   DATA[2295,34] := 2.0;
   DATA[2295,35] := 250.1762;
   DATA[2295,36] := 1.681991;
   DATA[2295,37] := 189.1022;
   DATA[2295,38] := 0.000128152;
   DATA[2295,39] := 1.0;
   DATA[2295,40] := 1.0;
   DATA[2296,0] := 2.444992;
   DATA[2296,1] := 865.3663;
   DATA[2296,2] := 2.0;
   DATA[2296,3] := 2.0;
   DATA[2296,4] := 262.3366;
   DATA[2296,5] := 8.395475;
   DATA[2296,6] := 330.0948;
   DATA[2296,7] := 2.455259;
   DATA[2296,8] := 2.0;
   DATA[2296,9] := 2.0;
   DATA[2296,10] := 2.0;
   DATA[2296,11] := 19.70037;
   DATA[2296,12] := 2.203632;
   DATA[2296,13] := 815.7364;
   DATA[2296,14] := 1.0;
   DATA[2296,15] := 2.0;
   DATA[2296,16] := 1.0;
   DATA[2296,17] := 1.0;
   DATA[2296,18] := 1.0;
   DATA[2296,19] := 2.0;
   DATA[2296,20] := 148.808;
   DATA[2296,21] := 155.0115;
   DATA[2296,22] := 1.714926;
   DATA[2296,23] := 851.2817;
   DATA[2296,24] := 2.0;
   DATA[2296,25] := 2.0;
   DATA[2296,26] := 7.873174;
   DATA[2296,27] := 144.3989;
   DATA[2296,28] := 261.7278;
   DATA[2296,29] := 11.95847;
   DATA[2296,30] := 1.723148;
   DATA[2296,31] := 1.281798;
   DATA[2296,32] := 0.7348846;
   DATA[2296,33] := 0.3083624;
   DATA[2296,34] := 2.0;
   DATA[2296,35] := 250.1762;
   DATA[2296,36] := 1.681991;
   DATA[2296,37] := 188.958;
   DATA[2296,38] := 0.000128152;
   DATA[2296,39] := 1.0;
   DATA[2296,40] := 1.0;
   DATA[2297,0] := 2.431861;
   DATA[2297,1] := 865.1308;
   DATA[2297,2] := 2.0;
   DATA[2297,3] := 2.0;
   DATA[2297,4] := 262.3366;
   DATA[2297,5] := 8.395475;
   DATA[2297,6] := 330.0948;
   DATA[2297,7] := 2.455259;
   DATA[2297,8] := 2.0;
   DATA[2297,9] := 2.0;
   DATA[2297,10] := 2.0;
   DATA[2297,11] := 19.70037;
   DATA[2297,12] := 2.203632;
   DATA[2297,13] := 815.456;
   DATA[2297,14] := 1.0;
   DATA[2297,15] := 2.0;
   DATA[2297,16] := 1.0;
   DATA[2297,17] := 1.0;
   DATA[2297,18] := 1.0;
   DATA[2297,19] := 2.0;
   DATA[2297,20] := 148.808;
   DATA[2297,21] := 155.0115;
   DATA[2297,22] := 1.714926;
   DATA[2297,23] := 851.2433;
   DATA[2297,24] := 2.0;
   DATA[2297,25] := 2.0;
   DATA[2297,26] := 7.873174;
   DATA[2297,27] := 144.3989;
   DATA[2297,28] := 261.7278;
   DATA[2297,29] := 11.95847;
   DATA[2297,30] := 1.723148;
   DATA[2297,31] := 1.304214;
   DATA[2297,32] := 0.7348846;
   DATA[2297,33] := 0.3083624;
   DATA[2297,34] := 2.0;
   DATA[2297,35] := 250.1762;
   DATA[2297,36] := 1.681991;
   DATA[2297,37] := 188.958;
   DATA[2297,38] := 0.000128152;
   DATA[2297,39] := 1.0;
   DATA[2297,40] := 1.0;
   DATA[2298,0] := 2.425776;
   DATA[2298,1] := 865.4056;
   DATA[2298,2] := 2.0;
   DATA[2298,3] := 2.0;
   DATA[2298,4] := 262.3366;
   DATA[2298,5] := 8.395475;
   DATA[2298,6] := 330.0948;
   DATA[2298,7] := 2.455259;
   DATA[2298,8] := 2.0;
   DATA[2298,9] := 2.0;
   DATA[2298,10] := 2.0;
   DATA[2298,11] := 19.70037;
   DATA[2298,12] := 2.203632;
   DATA[2298,13] := 815.6162;
   DATA[2298,14] := 1.0;
   DATA[2298,15] := 2.0;
   DATA[2298,16] := 1.0;
   DATA[2298,17] := 1.0;
   DATA[2298,18] := 1.0;
   DATA[2298,19] := 2.0;
   DATA[2298,20] := 148.808;
   DATA[2298,21] := 155.0115;
   DATA[2298,22] := 1.714926;
   DATA[2298,23] := 851.3971;
   DATA[2298,24] := 2.0;
   DATA[2298,25] := 2.0;
   DATA[2298,26] := 7.873174;
   DATA[2298,27] := 144.3989;
   DATA[2298,28] := 261.7278;
   DATA[2298,29] := 11.95847;
   DATA[2298,30] := 1.723148;
   DATA[2298,31] := 1.310747;
   DATA[2298,32] := 0.7348846;
   DATA[2298,33] := 0.3083624;
   DATA[2298,34] := 2.0;
   DATA[2298,35] := 250.1762;
   DATA[2298,36] := 1.681991;
   DATA[2298,37] := 188.958;
   DATA[2298,38] := 0.000128152;
   DATA[2298,39] := 1.0;
   DATA[2298,40] := 1.0;
   DATA[2299,0] := 2.425456;
   DATA[2299,1] := 865.5626;
   DATA[2299,2] := 2.0;
   DATA[2299,3] := 2.0;
   DATA[2299,4] := 262.3366;
   DATA[2299,5] := 8.395475;
   DATA[2299,6] := 330.0948;
   DATA[2299,7] := 2.456156;
   DATA[2299,8] := 2.0;
   DATA[2299,9] := 2.0;
   DATA[2299,10] := 2.0;
   DATA[2299,11] := 19.67796;
   DATA[2299,12] := 2.206322;
   DATA[2299,13] := 815.416;
   DATA[2299,14] := 1.0;
   DATA[2299,15] := 2.0;
   DATA[2299,16] := 1.0;
   DATA[2299,17] := 1.0;
   DATA[2299,18] := 1.0;
   DATA[2299,19] := 2.0;
   DATA[2299,20] := 148.808;
   DATA[2299,21] := 155.0115;
   DATA[2299,22] := 1.714926;
   DATA[2299,23] := 851.3971;
   DATA[2299,24] := 2.0;
   DATA[2299,25] := 2.0;
   DATA[2299,26] := 7.874776;
   DATA[2299,27] := 144.5014;
   DATA[2299,28] := 261.7278;
   DATA[2299,29] := 11.95847;
   DATA[2299,30] := 1.725327;
   DATA[2299,31] := 1.311772;
   DATA[2299,32] := 0.7348846;
   DATA[2299,33] := 0.3083624;
   DATA[2299,34] := 2.0;
   DATA[2299,35] := 250.1762;
   DATA[2299,36] := 1.681991;
   DATA[2299,37] := 188.958;
   DATA[2299,38] := 0.000128152;
   DATA[2299,39] := 1.0;
   DATA[2299,40] := 1.0;
   DATA[2300,0] := 2.451398;
   DATA[2300,1] := 865.7589;
   DATA[2300,2] := 2.0;
   DATA[2300,3] := 2.0;
   DATA[2300,4] := 262.3366;
   DATA[2300,5] := 8.395475;
   DATA[2300,6] := 330.0948;
   DATA[2300,7] := 2.456156;
   DATA[2300,8] := 2.0;
   DATA[2300,9] := 2.0;
   DATA[2300,10] := 2.0;
   DATA[2300,11] := 19.65235;
   DATA[2300,12] := 2.207091;
   DATA[2300,13] := 815.2157;
   DATA[2300,14] := 1.0;
   DATA[2300,15] := 2.0;
   DATA[2300,16] := 1.0;
   DATA[2300,17] := 1.0;
   DATA[2300,18] := 1.0;
   DATA[2300,19] := 2.0;
   DATA[2300,20] := 148.808;
   DATA[2300,21] := 155.0115;
   DATA[2300,22] := 1.717874;
   DATA[2300,23] := 851.7432;
   DATA[2300,24] := 2.0;
   DATA[2300,25] := 2.0;
   DATA[2300,26] := 7.874776;
   DATA[2300,27] := 144.5014;
   DATA[2300,28] := 261.7278;
   DATA[2300,29] := 11.95847;
   DATA[2300,30] := 1.725327;
   DATA[2300,31] := 1.312284;
   DATA[2300,32] := 0.7348846;
   DATA[2300,33] := 0.3083624;
   DATA[2300,34] := 2.0;
   DATA[2300,35] := 250.1762;
   DATA[2300,36] := 1.681991;
   DATA[2300,37] := 188.958;
   DATA[2300,38] := 0.000128152;
   DATA[2300,39] := 1.0;
   DATA[2300,40] := 1.0;
   DATA[2301,0] := 2.498479;
   DATA[2301,1] := 865.7981;
   DATA[2301,2] := 2.0;
   DATA[2301,3] := 2.0;
   DATA[2301,4] := 262.3366;
   DATA[2301,5] := 8.395475;
   DATA[2301,6] := 330.0948;
   DATA[2301,7] := 2.456156;
   DATA[2301,8] := 2.0;
   DATA[2301,9] := 2.0;
   DATA[2301,10] := 2.0;
   DATA[2301,11] := 19.65235;
   DATA[2301,12] := 2.207091;
   DATA[2301,13] := 814.8552;
   DATA[2301,14] := 1.0;
   DATA[2301,15] := 2.0;
   DATA[2301,16] := 1.0;
   DATA[2301,17] := 1.0;
   DATA[2301,18] := 1.0;
   DATA[2301,19] := 2.0;
   DATA[2301,20] := 148.808;
   DATA[2301,21] := 155.0884;
   DATA[2301,22] := 1.718515;
   DATA[2301,23] := 851.3971;
   DATA[2301,24] := 2.0;
   DATA[2301,25] := 2.0;
   DATA[2301,26] := 7.874776;
   DATA[2301,27] := 144.5014;
   DATA[2301,28] := 261.7278;
   DATA[2301,29] := 11.95847;
   DATA[2301,30] := 1.725711;
   DATA[2301,31] := 1.298578;
   DATA[2301,32] := 0.7353967;
   DATA[2301,33] := 0.3083624;
   DATA[2301,34] := 2.0;
   DATA[2301,35] := 250.1762;
   DATA[2301,36] := 1.681991;
   DATA[2301,37] := 188.958;
   DATA[2301,38] := 0.000128152;
   DATA[2301,39] := 1.0;
   DATA[2301,40] := 1.0;
   DATA[2302,0] := 2.539474;
   DATA[2302,1] := 866.1906;
   DATA[2302,2] := 2.0;
   DATA[2302,3] := 2.0;
   DATA[2302,4] := 262.3366;
   DATA[2302,5] := 8.395475;
   DATA[2302,6] := 330.0948;
   DATA[2302,7] := 2.456156;
   DATA[2302,8] := 2.0;
   DATA[2302,9] := 2.0;
   DATA[2302,10] := 2.0;
   DATA[2302,11] := 19.69396;
   DATA[2302,12] := 2.207091;
   DATA[2302,13] := 814.8552;
   DATA[2302,14] := 1.0;
   DATA[2302,15] := 2.0;
   DATA[2302,16] := 1.0;
   DATA[2302,17] := 1.0;
   DATA[2302,18] := 1.0;
   DATA[2302,19] := 2.0;
   DATA[2302,20] := 148.808;
   DATA[2302,21] := 155.0884;
   DATA[2302,22] := 1.718515;
   DATA[2302,23] := 851.3971;
   DATA[2302,24] := 2.0;
   DATA[2302,25] := 2.0;
   DATA[2302,26] := 7.874776;
   DATA[2302,27] := 144.5014;
   DATA[2302,28] := 261.7278;
   DATA[2302,29] := 11.95847;
   DATA[2302,30] := 1.727634;
   DATA[2302,31] := 1.292046;
   DATA[2302,32] := 0.7353967;
   DATA[2302,33] := 0.3083624;
   DATA[2302,34] := 2.0;
   DATA[2302,35] := 250.1762;
   DATA[2302,36] := 1.681991;
   DATA[2302,37] := 189.1022;
   DATA[2302,38] := 0.000128152;
   DATA[2302,39] := 1.0;
   DATA[2302,40] := 1.0;
   DATA[2303,0] := 2.580149;
   DATA[2303,1] := 865.7981;
   DATA[2303,2] := 2.0;
   DATA[2303,3] := 2.0;
   DATA[2303,4] := 262.3366;
   DATA[2303,5] := 8.395475;
   DATA[2303,6] := 330.0948;
   DATA[2303,7] := 2.457566;
   DATA[2303,8] := 2.0;
   DATA[2303,9] := 2.0;
   DATA[2303,10] := 2.0;
   DATA[2303,11] := 19.69396;
   DATA[2303,12] := 2.207091;
   DATA[2303,13] := 814.7751;
   DATA[2303,14] := 1.0;
   DATA[2303,15] := 2.0;
   DATA[2303,16] := 1.0;
   DATA[2303,17] := 1.0;
   DATA[2303,18] := 1.0;
   DATA[2303,19] := 2.0;
   DATA[2303,20] := 148.808;
   DATA[2303,21] := 155.0884;
   DATA[2303,22] := 1.718515;
   DATA[2303,23] := 852.0508;
   DATA[2303,24] := 2.0;
   DATA[2303,25] := 2.0;
   DATA[2303,26] := 7.874776;
   DATA[2303,27] := 144.5014;
   DATA[2303,28] := 261.7278;
   DATA[2303,29] := 11.95847;
   DATA[2303,30] := 1.727634;
   DATA[2303,31] := 1.300884;
   DATA[2303,32] := 0.7353967;
   DATA[2303,33] := 0.3083624;
   DATA[2303,34] := 2.0;
   DATA[2303,35] := 250.1762;
   DATA[2303,36] := 1.681991;
   DATA[2303,37] := 189.1662;
   DATA[2303,38] := 0.000128152;
   DATA[2303,39] := 1.0;
   DATA[2303,40] := 1.0;
   DATA[2304,0] := 2.620824;
   DATA[2304,1] := 865.9551;
   DATA[2304,2] := 2.0;
   DATA[2304,3] := 2.0;
   DATA[2304,4] := 262.3366;
   DATA[2304,5] := 8.395475;
   DATA[2304,6] := 330.0948;
   DATA[2304,7] := 2.457566;
   DATA[2304,8] := 2.0;
   DATA[2304,9] := 2.0;
   DATA[2304,10] := 2.0;
   DATA[2304,11] := 19.69396;
   DATA[2304,12] := 2.207091;
   DATA[2304,13] := 814.8151;
   DATA[2304,14] := 1.0;
   DATA[2304,15] := 2.0;
   DATA[2304,16] := 1.0;
   DATA[2304,17] := 1.0;
   DATA[2304,18] := 1.0;
   DATA[2304,19] := 2.0;
   DATA[2304,20] := 148.808;
   DATA[2304,21] := 155.0884;
   DATA[2304,22] := 1.718515;
   DATA[2304,23] := 852.4353;
   DATA[2304,24] := 2.0;
   DATA[2304,25] := 2.0;
   DATA[2304,26] := 7.874776;
   DATA[2304,27] := 144.5014;
   DATA[2304,28] := 261.7278;
   DATA[2304,29] := 11.95847;
   DATA[2304,30] := 1.727634;
   DATA[2304,31] := 1.305367;
   DATA[2304,32] := 0.7353967;
   DATA[2304,33] := 0.3083624;
   DATA[2304,34] := 2.0;
   DATA[2304,35] := 250.3044;
   DATA[2304,36] := 1.681991;
   DATA[2304,37] := 189.1662;
   DATA[2304,38] := 0.000128152;
   DATA[2304,39] := 1.0;
   DATA[2304,40] := 1.0;
   DATA[2305,0] := 2.641642;
   DATA[2305,1] := 865.9551;
   DATA[2305,2] := 2.0;
   DATA[2305,3] := 2.0;
   DATA[2305,4] := 262.3366;
   DATA[2305,5] := 8.395475;
   DATA[2305,6] := 330.0436;
   DATA[2305,7] := 2.457566;
   DATA[2305,8] := 2.0;
   DATA[2305,9] := 2.0;
   DATA[2305,10] := 2.0;
   DATA[2305,11] := 19.69396;
   DATA[2305,12] := 2.208372;
   DATA[2305,13] := 814.735;
   DATA[2305,14] := 1.0;
   DATA[2305,15] := 2.0;
   DATA[2305,16] := 1.0;
   DATA[2305,17] := 1.0;
   DATA[2305,18] := 1.0;
   DATA[2305,19] := 2.0;
   DATA[2305,20] := 148.808;
   DATA[2305,21] := 155.0884;
   DATA[2305,22] := 1.718515;
   DATA[2305,23] := 852.5506;
   DATA[2305,24] := 2.0;
   DATA[2305,25] := 2.0;
   DATA[2305,26] := 7.874455;
   DATA[2305,27] := 144.5014;
   DATA[2305,28] := 261.7278;
   DATA[2305,29] := 11.95847;
   DATA[2305,30] := 1.725455;
   DATA[2305,31] := 1.311003;
   DATA[2305,32] := 0.7353967;
   DATA[2305,33] := 0.3083624;
   DATA[2305,34] := 2.0;
   DATA[2305,35] := 250.3525;
   DATA[2305,36] := 1.681991;
   DATA[2305,37] := 189.1662;
   DATA[2305,38] := 0.000128152;
   DATA[2305,39] := 1.0;
   DATA[2305,40] := 1.0;
   DATA[2306,0] := 2.657016;
   DATA[2306,1] := 866.2691;
   DATA[2306,2] := 2.0;
   DATA[2306,3] := 2.0;
   DATA[2306,4] := 262.3366;
   DATA[2306,5] := 8.395475;
   DATA[2306,6] := 329.9667;
   DATA[2306,7] := 2.457566;
   DATA[2306,8] := 2.0;
   DATA[2306,9] := 2.0;
   DATA[2306,10] := 2.0;
   DATA[2306,11] := 19.69396;
   DATA[2306,12] := 2.208884;
   DATA[2306,13] := 815.0154;
   DATA[2306,14] := 1.0;
   DATA[2306,15] := 2.0;
   DATA[2306,16] := 1.0;
   DATA[2306,17] := 1.0;
   DATA[2306,18] := 1.0;
   DATA[2306,19] := 2.0;
   DATA[2306,20] := 148.808;
   DATA[2306,21] := 155.0884;
   DATA[2306,22] := 1.718515;
   DATA[2306,23] := 853.1274;
   DATA[2306,24] := 2.0;
   DATA[2306,25] := 2.0;
   DATA[2306,26] := 7.874455;
   DATA[2306,27] := 144.5014;
   DATA[2306,28] := 261.5355;
   DATA[2306,29] := 11.95847;
   DATA[2306,30] := 1.725455;
   DATA[2306,31] := 1.312284;
   DATA[2306,32] := 0.7353967;
   DATA[2306,33] := 0.3083624;
   DATA[2306,34] := 2.0;
   DATA[2306,35] := 250.3525;
   DATA[2306,36] := 1.681991;
   DATA[2306,37] := 189.1662;
   DATA[2306,38] := 0.000128152;
   DATA[2306,39] := 1.0;
   DATA[2306,40] := 1.0;
   DATA[2307,0] := 2.657336;
   DATA[2307,1] := 866.3083;
   DATA[2307,2] := 2.0;
   DATA[2307,3] := 2.0;
   DATA[2307,4] := 262.3366;
   DATA[2307,5] := 8.395475;
   DATA[2307,6] := 329.9667;
   DATA[2307,7] := 2.456541;
   DATA[2307,8] := 2.0;
   DATA[2307,9] := 2.0;
   DATA[2307,10] := 2.0;
   DATA[2307,11] := 19.69396;
   DATA[2307,12] := 2.208884;
   DATA[2307,13] := 814.4547;
   DATA[2307,14] := 1.0;
   DATA[2307,15] := 2.0;
   DATA[2307,16] := 1.0;
   DATA[2307,17] := 1.0;
   DATA[2307,18] := 1.0;
   DATA[2307,19] := 2.0;
   DATA[2307,20] := 148.808;
   DATA[2307,21] := 155.0884;
   DATA[2307,22] := 1.718515;
   DATA[2307,23] := 853.5119;
   DATA[2307,24] := 2.0;
   DATA[2307,25] := 2.0;
   DATA[2307,26] := 7.874455;
   DATA[2307,27] := 144.5014;
   DATA[2307,28] := 261.5355;
   DATA[2307,29] := 11.95847;
   DATA[2307,30] := 1.725455;
   DATA[2307,31] := 1.301012;
   DATA[2307,32] := 0.7353967;
   DATA[2307,33] := 0.3083624;
   DATA[2307,34] := 2.0;
   DATA[2307,35] := 250.3525;
   DATA[2307,36] := 1.681991;
   DATA[2307,37] := 189.1662;
   DATA[2307,38] := 0.000128152;
   DATA[2307,39] := 1.0;
   DATA[2307,40] := 1.0;
   DATA[2308,0] := 2.639721;
   DATA[2308,1] := 866.4654;
   DATA[2308,2] := 2.0;
   DATA[2308,3] := 2.0;
   DATA[2308,4] := 262.3366;
   DATA[2308,5] := 8.395475;
   DATA[2308,6] := 329.9667;
   DATA[2308,7] := 2.456541;
   DATA[2308,8] := 2.0;
   DATA[2308,9] := 2.0;
   DATA[2308,10] := 2.0;
   DATA[2308,11] := 19.69396;
   DATA[2308,12] := 2.208884;
   DATA[2308,13] := 814.735;
   DATA[2308,14] := 1.0;
   DATA[2308,15] := 2.0;
   DATA[2308,16] := 1.0;
   DATA[2308,17] := 1.0;
   DATA[2308,18] := 1.0;
   DATA[2308,19] := 2.0;
   DATA[2308,20] := 148.808;
   DATA[2308,21] := 155.0884;
   DATA[2308,22] := 1.717746;
   DATA[2308,23] := 853.3965;
   DATA[2308,24] := 2.0;
   DATA[2308,25] := 2.0;
   DATA[2308,26] := 7.874135;
   DATA[2308,27] := 144.5014;
   DATA[2308,28] := 261.5355;
   DATA[2308,29] := 11.95847;
   DATA[2308,30] := 1.725455;
   DATA[2308,31] := 1.29243;
   DATA[2308,32] := 0.7353967;
   DATA[2308,33] := 0.3083624;
   DATA[2308,34] := 2.0;
   DATA[2308,35] := 250.3525;
   DATA[2308,36] := 1.681991;
   DATA[2308,37] := 189.1662;
   DATA[2308,38] := 0.000128152;
   DATA[2308,39] := 1.0;
   DATA[2308,40] := 1.0;
   DATA[2309,0] := 2.624347;
   DATA[2309,1] := 866.1906;
   DATA[2309,2] := 2.0;
   DATA[2309,3] := 2.0;
   DATA[2309,4] := 262.3366;
   DATA[2309,5] := 8.395475;
   DATA[2309,6] := 329.9667;
   DATA[2309,7] := 2.456541;
   DATA[2309,8] := 2.0;
   DATA[2309,9] := 2.0;
   DATA[2309,10] := 2.0;
   DATA[2309,11] := 19.72598;
   DATA[2309,12] := 2.209653;
   DATA[2309,13] := 814.2143;
   DATA[2309,14] := 1.0;
   DATA[2309,15] := 2.0;
   DATA[2309,16] := 1.0;
   DATA[2309,17] := 1.0;
   DATA[2309,18] := 1.0;
   DATA[2309,19] := 2.0;
   DATA[2309,20] := 148.808;
   DATA[2309,21] := 155.0884;
   DATA[2309,22] := 1.71608;
   DATA[2309,23] := 853.858;
   DATA[2309,24] := 2.0;
   DATA[2309,25] := 2.0;
   DATA[2309,26] := 7.874135;
   DATA[2309,27] := 144.5014;
   DATA[2309,28] := 261.5355;
   DATA[2309,29] := 11.95847;
   DATA[2309,30] := 1.725455;
   DATA[2309,31] := 1.292174;
   DATA[2309,32] := 0.7353967;
   DATA[2309,33] := 0.3083624;
   DATA[2309,34] := 2.0;
   DATA[2309,35] := 250.2403;
   DATA[2309,36] := 1.681991;
   DATA[2309,37] := 189.0381;
   DATA[2309,38] := 0.000128152;
   DATA[2309,39] := 1.0;
   DATA[2309,40] := 1.0;
   DATA[2310,0] := 2.618582;
   DATA[2310,1] := 866.5831;
   DATA[2310,2] := 2.0;
   DATA[2310,3] := 2.0;
   DATA[2310,4] := 262.3366;
   DATA[2310,5] := 8.395475;
   DATA[2310,6] := 329.9667;
   DATA[2310,7] := 2.456541;
   DATA[2310,8] := 2.0;
   DATA[2310,9] := 2.0;
   DATA[2310,10] := 2.0;
   DATA[2310,11] := 19.73238;
   DATA[2310,12] := 2.210166;
   DATA[2310,13] := 814.6149;
   DATA[2310,14] := 1.0;
   DATA[2310,15] := 2.0;
   DATA[2310,16] := 1.0;
   DATA[2310,17] := 1.0;
   DATA[2310,18] := 1.0;
   DATA[2310,19] := 2.0;
   DATA[2310,20] := 148.808;
   DATA[2310,21] := 155.0884;
   DATA[2310,22] := 1.715952;
   DATA[2310,23] := 853.7811;
   DATA[2310,24] := 2.0;
   DATA[2310,25] := 2.0;
   DATA[2310,26] := 7.874135;
   DATA[2310,27] := 144.5014;
   DATA[2310,28] := 261.5355;
   DATA[2310,29] := 11.95847;
   DATA[2310,30] := 1.725455;
   DATA[2310,31] := 1.292174;
   DATA[2310,32] := 0.7353967;
   DATA[2310,33] := 0.3083624;
   DATA[2310,34] := 2.0;
   DATA[2310,35] := 250.2403;
   DATA[2310,36] := 1.681991;
   DATA[2310,37] := 189.0381;
   DATA[2310,38] := 0.000128152;
   DATA[2310,39] := 1.0;
   DATA[2310,40] := 1.0;
   DATA[2311,0] := 2.612818;
   DATA[2311,1] := 866.1121;
   DATA[2311,2] := 2.0;
   DATA[2311,3] := 2.0;
   DATA[2311,4] := 262.3366;
   DATA[2311,5] := 8.395475;
   DATA[2311,6] := 329.9667;
   DATA[2311,7] := 2.456541;
   DATA[2311,8] := 2.0;
   DATA[2311,9] := 2.0;
   DATA[2311,10] := 2.0;
   DATA[2311,11] := 19.66835;
   DATA[2311,12] := 2.210166;
   DATA[2311,13] := 814.4547;
   DATA[2311,14] := 1.0;
   DATA[2311,15] := 2.0;
   DATA[2311,16] := 1.0;
   DATA[2311,17] := 1.0;
   DATA[2311,18] := 1.0;
   DATA[2311,19] := 2.0;
   DATA[2311,20] := 148.808;
   DATA[2311,21] := 155.0884;
   DATA[2311,22] := 1.715952;
   DATA[2311,23] := 854.1271;
   DATA[2311,24] := 2.0;
   DATA[2311,25] := 2.0;
   DATA[2311,26] := 7.874135;
   DATA[2311,27] := 144.5014;
   DATA[2311,28] := 261.5996;
   DATA[2311,29] := 11.95847;
   DATA[2311,30] := 1.725455;
   DATA[2311,31] := 1.292174;
   DATA[2311,32] := 0.7353967;
   DATA[2311,33] := 0.3083624;
   DATA[2311,34] := 2.0;
   DATA[2311,35] := 250.2403;
   DATA[2311,36] := 1.681991;
   DATA[2311,37] := 189.0381;
   DATA[2311,38] := 0.000128152;
   DATA[2311,39] := 1.0;
   DATA[2311,40] := 1.0;
   DATA[2312,0] := 2.598405;
   DATA[2312,1] := 865.6803;
   DATA[2312,2] := 2.0;
   DATA[2312,3] := 2.0;
   DATA[2312,4] := 262.3366;
   DATA[2312,5] := 8.395475;
   DATA[2312,6] := 329.9667;
   DATA[2312,7] := 2.456541;
   DATA[2312,8] := 2.0;
   DATA[2312,9] := 2.0;
   DATA[2312,10] := 2.0;
   DATA[2312,11] := 19.62994;
   DATA[2312,12] := 2.210166;
   DATA[2312,13] := 814.7751;
   DATA[2312,14] := 1.0;
   DATA[2312,15] := 2.0;
   DATA[2312,16] := 1.0;
   DATA[2312,17] := 1.0;
   DATA[2312,18] := 1.0;
   DATA[2312,19] := 2.0;
   DATA[2312,20] := 148.808;
   DATA[2312,21] := 155.0884;
   DATA[2312,22] := 1.715952;
   DATA[2312,23] := 854.2425;
   DATA[2312,24] := 2.0;
   DATA[2312,25] := 2.0;
   DATA[2312,26] := 7.874135;
   DATA[2312,27] := 144.5014;
   DATA[2312,28] := 261.8239;
   DATA[2312,29] := 11.95847;
   DATA[2312,30] := 1.725455;
   DATA[2312,31] := 1.300115;
   DATA[2312,32] := 0.7353967;
   DATA[2312,33] := 0.3083624;
   DATA[2312,34] := 2.0;
   DATA[2312,35] := 250.2403;
   DATA[2312,36] := 1.681991;
   DATA[2312,37] := 189.0381;
   DATA[2312,38] := 0.000128152;
   DATA[2312,39] := 1.0;
   DATA[2312,40] := 1.0;
   DATA[2313,0] := 2.582071;
   DATA[2313,1] := 865.6803;
   DATA[2313,2] := 2.0;
   DATA[2313,3] := 2.0;
   DATA[2313,4] := 262.3366;
   DATA[2313,5] := 8.395475;
   DATA[2313,6] := 330.1718;
   DATA[2313,7] := 2.456541;
   DATA[2313,8] := 2.0;
   DATA[2313,9] := 2.0;
   DATA[2313,10] := 2.0;
   DATA[2313,11] := 19.62994;
   DATA[2313,12] := 2.210166;
   DATA[2313,13] := 814.6149;
   DATA[2313,14] := 1.0;
   DATA[2313,15] := 2.0;
   DATA[2313,16] := 1.0;
   DATA[2313,17] := 1.0;
   DATA[2313,18] := 1.0;
   DATA[2313,19] := 2.0;
   DATA[2313,20] := 148.808;
   DATA[2313,21] := 155.0884;
   DATA[2313,22] := 1.715952;
   DATA[2313,23] := 854.4732;
   DATA[2313,24] := 2.0;
   DATA[2313,25] := 2.0;
   DATA[2313,26] := 7.874135;
   DATA[2313,27] := 144.5014;
   DATA[2313,28] := 261.8239;
   DATA[2313,29] := 11.95847;
   DATA[2313,30] := 1.725455;
   DATA[2313,31] := 1.297041;
   DATA[2313,32] := 0.7353967;
   DATA[2313,33] := 0.3083624;
   DATA[2313,34] := 2.0;
   DATA[2313,35] := 250.1122;
   DATA[2313,36] := 1.681991;
   DATA[2313,37] := 189.0381;
   DATA[2313,38] := 0.000128152;
   DATA[2313,39] := 1.0;
   DATA[2313,40] := 1.0;
   DATA[2314,0] := 2.564456;
   DATA[2314,1] := 865.7981;
   DATA[2314,2] := 2.0;
   DATA[2314,3] := 2.0;
   DATA[2314,4] := 262.3366;
   DATA[2314,5] := 8.395475;
   DATA[2314,6] := 330.1718;
   DATA[2314,7] := 2.456541;
   DATA[2314,8] := 2.0;
   DATA[2314,9] := 2.0;
   DATA[2314,10] := 2.0;
   DATA[2314,11] := 19.62994;
   DATA[2314,12] := 2.210166;
   DATA[2314,13] := 814.9353;
   DATA[2314,14] := 1.0;
   DATA[2314,15] := 2.0;
   DATA[2314,16] := 1.0;
   DATA[2314,17] := 1.0;
   DATA[2314,18] := 1.0;
   DATA[2314,19] := 2.0;
   DATA[2314,20] := 148.808;
   DATA[2314,21] := 155.0884;
   DATA[2314,22] := 1.715952;
   DATA[2314,23] := 854.5501;
   DATA[2314,24] := 2.0;
   DATA[2314,25] := 2.0;
   DATA[2314,26] := 7.874135;
   DATA[2314,27] := 144.5014;
   DATA[2314,28] := 261.8239;
   DATA[2314,29] := 11.95847;
   DATA[2314,30] := 1.725455;
   DATA[2314,31] := 1.301652;
   DATA[2314,32] := 0.7353967;
   DATA[2314,33] := 0.3083624;
   DATA[2314,34] := 2.0;
   DATA[2314,35] := 250.1122;
   DATA[2314,36] := 1.681991;
   DATA[2314,37] := 189.0381;
   DATA[2314,38] := 0.000128152;
   DATA[2314,39] := 1.0;
   DATA[2314,40] := 1.0;
   DATA[2315,0] := 2.551324;
   DATA[2315,1] := 865.9943;
   DATA[2315,2] := 2.0;
   DATA[2315,3] := 2.0;
   DATA[2315,4] := 262.3366;
   DATA[2315,5] := 8.395475;
   DATA[2315,6] := 330.1718;
   DATA[2315,7] := 2.456541;
   DATA[2315,8] := 2.0;
   DATA[2315,9] := 2.0;
   DATA[2315,10] := 2.0;
   DATA[2315,11] := 19.67476;
   DATA[2315,12] := 2.210166;
   DATA[2315,13] := 814.7751;
   DATA[2315,14] := 1.0;
   DATA[2315,15] := 2.0;
   DATA[2315,16] := 1.0;
   DATA[2315,17] := 1.0;
   DATA[2315,18] := 1.0;
   DATA[2315,19] := 2.0;
   DATA[2315,20] := 148.808;
   DATA[2315,21] := 155.0884;
   DATA[2315,22] := 1.715952;
   DATA[2315,23] := 854.4732;
   DATA[2315,24] := 2.0;
   DATA[2315,25] := 2.0;
   DATA[2315,26] := 7.874135;
   DATA[2315,27] := 144.5014;
   DATA[2315,28] := 261.8239;
   DATA[2315,29] := 11.95847;
   DATA[2315,30] := 1.725455;
   DATA[2315,31] := 1.301652;
   DATA[2315,32] := 0.7353967;
   DATA[2315,33] := 0.3083624;
   DATA[2315,34] := 2.0;
   DATA[2315,35] := 250.1122;
   DATA[2315,36] := 1.681991;
   DATA[2315,37] := 189.0381;
   DATA[2315,38] := 0.000128152;
   DATA[2315,39] := 1.0;
   DATA[2315,40] := 1.0;
   DATA[2316,0] := 2.532428;
   DATA[2316,1] := 866.0729;
   DATA[2316,2] := 2.0;
   DATA[2316,3] := 2.0;
   DATA[2316,4] := 262.3366;
   DATA[2316,5] := 8.395475;
   DATA[2316,6] := 330.1718;
   DATA[2316,7] := 2.456541;
   DATA[2316,8] := 2.0;
   DATA[2316,9] := 2.0;
   DATA[2316,10] := 2.0;
   DATA[2316,11] := 19.67476;
   DATA[2316,12] := 2.208756;
   DATA[2316,13] := 815.3759;
   DATA[2316,14] := 1.0;
   DATA[2316,15] := 2.0;
   DATA[2316,16] := 1.0;
   DATA[2316,17] := 1.0;
   DATA[2316,18] := 1.0;
   DATA[2316,19] := 2.0;
   DATA[2316,20] := 148.808;
   DATA[2316,21] := 155.1653;
   DATA[2316,22] := 1.716721;
   DATA[2316,23] := 854.7039;
   DATA[2316,24] := 2.0;
   DATA[2316,25] := 2.0;
   DATA[2316,26] := 7.874135;
   DATA[2316,27] := 144.5014;
   DATA[2316,28] := 261.8239;
   DATA[2316,29] := 11.95847;
   DATA[2316,30] := 1.724173;
   DATA[2316,31] := 1.306136;
   DATA[2316,32] := 0.7353967;
   DATA[2316,33] := 0.3083624;
   DATA[2316,34] := 2.0;
   DATA[2316,35] := 250.1122;
   DATA[2316,36] := 1.681991;
   DATA[2316,37] := 188.8939;
   DATA[2316,38] := 0.000128152;
   DATA[2316,39] := 1.0;
   DATA[2316,40] := 1.0;
   DATA[2317,0] := 2.510649;
   DATA[2317,1] := 865.6018;
   DATA[2317,2] := 2.0;
   DATA[2317,3] := 2.0;
   DATA[2317,4] := 262.3366;
   DATA[2317,5] := 8.395475;
   DATA[2317,6] := 330.0179;
   DATA[2317,7] := 2.456541;
   DATA[2317,8] := 2.0;
   DATA[2317,9] := 2.0;
   DATA[2317,10] := 2.0;
   DATA[2317,11] := 19.67476;
   DATA[2317,12] := 2.208756;
   DATA[2317,13] := 815.416;
   DATA[2317,14] := 1.0;
   DATA[2317,15] := 2.0;
   DATA[2317,16] := 1.0;
   DATA[2317,17] := 1.0;
   DATA[2317,18] := 1.0;
   DATA[2317,19] := 2.0;
   DATA[2317,20] := 148.808;
   DATA[2317,21] := 155.1653;
   DATA[2317,22] := 1.716721;
   DATA[2317,23] := 854.627;
   DATA[2317,24] := 2.0;
   DATA[2317,25] := 2.0;
   DATA[2317,26] := 7.874135;
   DATA[2317,27] := 144.5014;
   DATA[2317,28] := 261.8239;
   DATA[2317,29] := 11.95847;
   DATA[2317,30] := 1.724173;
   DATA[2317,31] := 1.31254;
   DATA[2317,32] := 0.7353967;
   DATA[2317,33] := 0.3083624;
   DATA[2317,34] := 2.0;
   DATA[2317,35] := 250.0961;
   DATA[2317,36] := 1.681991;
   DATA[2317,37] := 188.7657;
   DATA[2317,38] := 0.000128152;
   DATA[2317,39] := 1.0;
   DATA[2317,40] := 1.0;
   DATA[2318,0] := 2.499439;
   DATA[2318,1] := 865.7589;
   DATA[2318,2] := 2.0;
   DATA[2318,3] := 2.0;
   DATA[2318,4] := 262.3366;
   DATA[2318,5] := 8.395475;
   DATA[2318,6] := 330.0179;
   DATA[2318,7] := 2.456541;
   DATA[2318,8] := 2.0;
   DATA[2318,9] := 2.0;
   DATA[2318,10] := 2.0;
   DATA[2318,11] := 19.67796;
   DATA[2318,12] := 2.208756;
   DATA[2318,13] := 815.3358;
   DATA[2318,14] := 1.0;
   DATA[2318,15] := 2.0;
   DATA[2318,16] := 1.0;
   DATA[2318,17] := 1.0;
   DATA[2318,18] := 1.0;
   DATA[2318,19] := 2.0;
   DATA[2318,20] := 148.808;
   DATA[2318,21] := 155.1653;
   DATA[2318,22] := 1.716721;
   DATA[2318,23] := 854.6655;
   DATA[2318,24] := 2.0;
   DATA[2318,25] := 2.0;
   DATA[2318,26] := 7.874135;
   DATA[2318,27] := 144.5014;
   DATA[2318,28] := 261.8239;
   DATA[2318,29] := 11.95847;
   DATA[2318,30] := 1.724173;
   DATA[2318,31] := 1.296016;
   DATA[2318,32] := 0.7353967;
   DATA[2318,33] := 0.3083624;
   DATA[2318,34] := 2.0;
   DATA[2318,35] := 249.984;
   DATA[2318,36] := 1.681991;
   DATA[2318,37] := 188.7657;
   DATA[2318,38] := 0.000128152;
   DATA[2318,39] := 1.0;
   DATA[2318,40] := 1.0;
   DATA[2319,0] := 2.480863;
   DATA[2319,1] := 865.4841;
   DATA[2319,2] := 2.0;
   DATA[2319,3] := 2.0;
   DATA[2319,4] := 262.3366;
   DATA[2319,5] := 8.395475;
   DATA[2319,6] := 330.0179;
   DATA[2319,7] := 2.456541;
   DATA[2319,8] := 2.0;
   DATA[2319,9] := 2.0;
   DATA[2319,10] := 2.0;
   DATA[2319,11] := 19.73238;
   DATA[2319,12] := 2.208756;
   DATA[2319,13] := 815.416;
   DATA[2319,14] := 1.0;
   DATA[2319,15] := 2.0;
   DATA[2319,16] := 1.0;
   DATA[2319,17] := 1.0;
   DATA[2319,18] := 1.0;
   DATA[2319,19] := 2.0;
   DATA[2319,20] := 148.808;
   DATA[2319,21] := 155.1653;
   DATA[2319,22] := 1.714286;
   DATA[2319,23] := 854.9346;
   DATA[2319,24] := 2.0;
   DATA[2319,25] := 2.0;
   DATA[2319,26] := 7.874135;
   DATA[2319,27] := 144.5014;
   DATA[2319,28] := 261.5675;
   DATA[2319,29] := 11.95847;
   DATA[2319,30] := 1.724173;
   DATA[2319,31] := 1.286153;
   DATA[2319,32] := 0.7353967;
   DATA[2319,33] := 0.3083624;
   DATA[2319,34] := 2.0;
   DATA[2319,35] := 249.8398;
   DATA[2319,36] := 1.681991;
   DATA[2319,37] := 188.6055;
   DATA[2319,38] := 0.000128152;
   DATA[2319,39] := 1.0;
   DATA[2319,40] := 1.0;
   DATA[2320,0] := 2.46581;
   DATA[2320,1] := 865.7981;
   DATA[2320,2] := 2.0;
   DATA[2320,3] := 2.0;
   DATA[2320,4] := 262.3366;
   DATA[2320,5] := 8.395475;
   DATA[2320,6] := 330.0179;
   DATA[2320,7] := 2.456541;
   DATA[2320,8] := 2.0;
   DATA[2320,9] := 2.0;
   DATA[2320,10] := 2.0;
   DATA[2320,11] := 19.73878;
   DATA[2320,12] := 2.208756;
   DATA[2320,13] := 815.456;
   DATA[2320,14] := 1.0;
   DATA[2320,15] := 2.0;
   DATA[2320,16] := 1.0;
   DATA[2320,17] := 1.0;
   DATA[2320,18] := 1.0;
   DATA[2320,19] := 2.0;
   DATA[2320,20] := 148.808;
   DATA[2320,21] := 155.1653;
   DATA[2320,22] := 1.711466;
   DATA[2320,23] := 855.0884;
   DATA[2320,24] := 2.0;
   DATA[2320,25] := 2.0;
   DATA[2320,26] := 7.874135;
   DATA[2320,27] := 144.5014;
   DATA[2320,28] := 261.5675;
   DATA[2320,29] := 11.95847;
   DATA[2320,30] := 1.724173;
   DATA[2320,31] := 1.288715;
   DATA[2320,32] := 0.7353967;
   DATA[2320,33] := 0.3083624;
   DATA[2320,34] := 2.0;
   DATA[2320,35] := 249.6956;
   DATA[2320,36] := 1.601897;
   DATA[2320,37] := 188.5734;
   DATA[2320,38] := 0.000128152;
   DATA[2320,39] := 1.0;
   DATA[2320,40] := 1.0;
   DATA[2321,0] := 2.451078;
   DATA[2321,1] := 865.5626;
   DATA[2321,2] := 2.0;
   DATA[2321,3] := 2.0;
   DATA[2321,4] := 262.3366;
   DATA[2321,5] := 8.395475;
   DATA[2321,6] := 330.0179;
   DATA[2321,7] := 2.456541;
   DATA[2321,8] := 2.0;
   DATA[2321,9] := 2.0;
   DATA[2321,10] := 2.0;
   DATA[2321,11] := 19.73878;
   DATA[2321,12] := 2.208756;
   DATA[2321,13] := 815.6162;
   DATA[2321,14] := 1.0;
   DATA[2321,15] := 2.0;
   DATA[2321,16] := 1.0;
   DATA[2321,17] := 1.0;
   DATA[2321,18] := 1.0;
   DATA[2321,19] := 2.0;
   DATA[2321,20] := 148.808;
   DATA[2321,21] := 155.1653;
   DATA[2321,22] := 1.711466;
   DATA[2321,23] := 855.5499;
   DATA[2321,24] := 2.0;
   DATA[2321,25] := 2.0;
   DATA[2321,26] := 7.874135;
   DATA[2321,27] := 144.5014;
   DATA[2321,28] := 261.5675;
   DATA[2321,29] := 11.95847;
   DATA[2321,30] := 1.722892;
   DATA[2321,31] := 1.282439;
   DATA[2321,32] := 0.7353967;
   DATA[2321,33] := 0.3083624;
   DATA[2321,34] := 2.0;
   DATA[2321,35] := 249.6956;
   DATA[2321,36] := 1.601897;
   DATA[2321,37] := 188.5734;
   DATA[2321,38] := 0.000128152;
   DATA[2321,39] := 1.0;
   DATA[2321,40] := 1.0;
   DATA[2322,0] := 2.439227;
   DATA[2322,1] := 865.2093;
   DATA[2322,2] := 2.0;
   DATA[2322,3] := 2.0;
   DATA[2322,4] := 262.3366;
   DATA[2322,5] := 8.395475;
   DATA[2322,6] := 330.0179;
   DATA[2322,7] := 2.456541;
   DATA[2322,8] := 2.0;
   DATA[2322,9] := 2.0;
   DATA[2322,10] := 2.0;
   DATA[2322,11] := 19.73878;
   DATA[2322,12] := 2.209013;
   DATA[2322,13] := 815.5361;
   DATA[2322,14] := 1.0;
   DATA[2322,15] := 2.0;
   DATA[2322,16] := 1.0;
   DATA[2322,17] := 1.0;
   DATA[2322,18] := 1.0;
   DATA[2322,19] := 2.0;
   DATA[2322,20] := 148.808;
   DATA[2322,21] := 155.1653;
   DATA[2322,22] := 1.711466;
   DATA[2322,23] := 855.4345;
   DATA[2322,24] := 2.0;
   DATA[2322,25] := 2.0;
   DATA[2322,26] := 7.874135;
   DATA[2322,27] := 144.5014;
   DATA[2322,28] := 261.5675;
   DATA[2322,29] := 11.95847;
   DATA[2322,30] := 1.721866;
   DATA[2322,31] := 1.282183;
   DATA[2322,32] := 0.7353967;
   DATA[2322,33] := 0.3083624;
   DATA[2322,34] := 2.0;
   DATA[2322,35] := 249.6956;
   DATA[2322,36] := 1.601897;
   DATA[2322,37] := 188.5734;
   DATA[2322,38] := 0.000128152;
   DATA[2322,39] := 1.0;
   DATA[2322,40] := 1.0;
   DATA[2323,0] := 2.426737;
   DATA[2323,1] := 865.3663;
   DATA[2323,2] := 2.0;
   DATA[2323,3] := 2.0;
   DATA[2323,4] := 262.3366;
   DATA[2323,5] := 8.395475;
   DATA[2323,6] := 330.0179;
   DATA[2323,7] := 2.454362;
   DATA[2323,8] := 2.0;
   DATA[2323,9] := 2.0;
   DATA[2323,10] := 2.0;
   DATA[2323,11] := 19.73878;
   DATA[2323,12] := 2.210166;
   DATA[2323,13] := 815.6563;
   DATA[2323,14] := 1.0;
   DATA[2323,15] := 2.0;
   DATA[2323,16] := 1.0;
   DATA[2323,17] := 1.0;
   DATA[2323,18] := 1.0;
   DATA[2323,19] := 2.0;
   DATA[2323,20] := 148.808;
   DATA[2323,21] := 155.1653;
   DATA[2323,22] := 1.71262;
   DATA[2323,23] := 855.473;
   DATA[2323,24] := 2.0;
   DATA[2323,25] := 2.0;
   DATA[2323,26] := 7.874135;
   DATA[2323,27] := 144.5014;
   DATA[2323,28] := 261.7278;
   DATA[2323,29] := 11.95847;
   DATA[2323,30] := 1.721866;
   DATA[2323,31] := 1.275906;
   DATA[2323,32] := 0.7353967;
   DATA[2323,33] := 0.3083624;
   DATA[2323,34] := 2.0;
   DATA[2323,35] := 249.9039;
   DATA[2323,36] := 1.601897;
   DATA[2323,37] := 188.5734;
   DATA[2323,38] := 0.000128152;
   DATA[2323,39] := 1.0;
   DATA[2323,40] := 1.0;
   DATA[2324,0] := 2.426416;
   DATA[2324,1] := 865.6803;
   DATA[2324,2] := 2.0;
   DATA[2324,3] := 2.0;
   DATA[2324,4] := 262.3366;
   DATA[2324,5] := 8.395475;
   DATA[2324,6] := 329.9667;
   DATA[2324,7] := 2.454234;
   DATA[2324,8] := 2.0;
   DATA[2324,9] := 2.0;
   DATA[2324,10] := 2.0;
   DATA[2324,11] := 19.83802;
   DATA[2324,12] := 2.210166;
   DATA[2324,13] := 815.1356;
   DATA[2324,14] := 1.0;
   DATA[2324,15] := 2.0;
   DATA[2324,16] := 1.0;
   DATA[2324,17] := 1.0;
   DATA[2324,18] := 1.0;
   DATA[2324,19] := 2.0;
   DATA[2324,20] := 148.808;
   DATA[2324,21] := 155.1653;
   DATA[2324,22] := 1.712876;
   DATA[2324,23] := 855.7421;
   DATA[2324,24] := 2.0;
   DATA[2324,25] := 2.0;
   DATA[2324,26] := 7.874135;
   DATA[2324,27] := 144.5014;
   DATA[2324,28] := 261.7278;
   DATA[2324,29] := 11.95847;
   DATA[2324,30] := 1.721866;
   DATA[2324,31] := 1.272832;
   DATA[2324,32] := 0.7353967;
   DATA[2324,33] := 0.3083624;
   DATA[2324,34] := 2.0;
   DATA[2324,35] := 249.9039;
   DATA[2324,36] := 1.601897;
   DATA[2324,37] := 188.5734;
   DATA[2324,38] := 0.000128152;
   DATA[2324,39] := 1.0;
   DATA[2324,40] := 1.0;
   DATA[2325,0] := 2.434744;
   DATA[2325,1] := 865.4841;
   DATA[2325,2] := 2.0;
   DATA[2325,3] := 2.0;
   DATA[2325,4] := 262.3366;
   DATA[2325,5] := 8.395475;
   DATA[2325,6] := 329.8898;
   DATA[2325,7] := 2.452952;
   DATA[2325,8] := 2.0;
   DATA[2325,9] := 2.0;
   DATA[2325,10] := 2.0;
   DATA[2325,11] := 19.85082;
   DATA[2325,12] := 2.210166;
   DATA[2325,13] := 815.0154;
   DATA[2325,14] := 1.0;
   DATA[2325,15] := 2.0;
   DATA[2325,16] := 1.0;
   DATA[2325,17] := 1.0;
   DATA[2325,18] := 1.0;
   DATA[2325,19] := 2.0;
   DATA[2325,20] := 148.808;
   DATA[2325,21] := 155.1653;
   DATA[2325,22] := 1.712876;
   DATA[2325,23] := 855.5499;
   DATA[2325,24] := 2.0;
   DATA[2325,25] := 2.0;
   DATA[2325,26] := 7.874135;
   DATA[2325,27] := 144.3989;
   DATA[2325,28] := 261.7278;
   DATA[2325,29] := 11.95847;
   DATA[2325,30] := 1.721866;
   DATA[2325,31] := 1.281542;
   DATA[2325,32] := 0.7353967;
   DATA[2325,33] := 0.3083624;
   DATA[2325,34] := 2.0;
   DATA[2325,35] := 249.9039;
   DATA[2325,36] := 1.601897;
   DATA[2325,37] := 188.5734;
   DATA[2325,38] := 0.000128152;
   DATA[2325,39] := 1.0;
   DATA[2325,40] := 1.0;
   DATA[2326,0] := 2.469013;
   DATA[2326,1] := 865.8766;
   DATA[2326,2] := 2.0;
   DATA[2326,3] := 2.0;
   DATA[2326,4] := 262.3366;
   DATA[2326,5] := 8.395475;
   DATA[2326,6] := 329.8898;
   DATA[2326,7] := 2.452952;
   DATA[2326,8] := 2.0;
   DATA[2326,9] := 2.0;
   DATA[2326,10] := 2.0;
   DATA[2326,11] := 19.85082;
   DATA[2326,12] := 2.210166;
   DATA[2326,13] := 814.9753;
   DATA[2326,14] := 1.0;
   DATA[2326,15] := 2.0;
   DATA[2326,16] := 1.0;
   DATA[2326,17] := 1.0;
   DATA[2326,18] := 1.0;
   DATA[2326,19] := 2.0;
   DATA[2326,20] := 148.808;
   DATA[2326,21] := 155.1653;
   DATA[2326,22] := 1.713901;
   DATA[2326,23] := 855.6268;
   DATA[2326,24] := 2.0;
   DATA[2326,25] := 2.0;
   DATA[2326,26] := 7.874135;
   DATA[2326,27] := 144.3989;
   DATA[2326,28] := 261.7278;
   DATA[2326,29] := 11.95847;
   DATA[2326,30] := 1.722507;
   DATA[2326,31] := 1.290509;
   DATA[2326,32] := 0.7353967;
   DATA[2326,33] := 0.3083624;
   DATA[2326,34] := 2.0;
   DATA[2326,35] := 249.9039;
   DATA[2326,36] := 1.730048;
   DATA[2326,37] := 188.8138;
   DATA[2326,38] := 0.000128152;
   DATA[2326,39] := 1.0;
   DATA[2326,40] := 1.0;
   DATA[2327,0] := 2.521218;
   DATA[2327,1] := 865.7589;
   DATA[2327,2] := 2.0;
   DATA[2327,3] := 2.0;
   DATA[2327,4] := 262.3366;
   DATA[2327,5] := 8.395475;
   DATA[2327,6] := 329.8898;
   DATA[2327,7] := 2.453593;
   DATA[2327,8] := 2.0;
   DATA[2327,9] := 2.0;
   DATA[2327,10] := 2.0;
   DATA[2327,11] := 19.85082;
   DATA[2327,12] := 2.210166;
   DATA[2327,13] := 814.9353;
   DATA[2327,14] := 1.0;
   DATA[2327,15] := 2.0;
   DATA[2327,16] := 1.0;
   DATA[2327,17] := 1.0;
   DATA[2327,18] := 1.0;
   DATA[2327,19] := 2.0;
   DATA[2327,20] := 148.808;
   DATA[2327,21] := 155.1653;
   DATA[2327,22] := 1.715311;
   DATA[2327,23] := 855.4345;
   DATA[2327,24] := 2.0;
   DATA[2327,25] := 2.0;
   DATA[2327,26] := 7.874135;
   DATA[2327,27] := 144.3989;
   DATA[2327,28] := 261.7278;
   DATA[2327,29] := 11.95847;
   DATA[2327,30] := 1.72302;
   DATA[2327,31] := 1.290893;
   DATA[2327,32] := 0.7353967;
   DATA[2327,33] := 0.3083624;
   DATA[2327,34] := 2.0;
   DATA[2327,35] := 249.9199;
   DATA[2327,36] := 1.730048;
   DATA[2327,37] := 188.8138;
   DATA[2327,38] := 0.000128152;
   DATA[2327,39] := 1.0;
   DATA[2327,40] := 1.0;
   DATA[2328,0] := 2.553246;
   DATA[2328,1] := 866.1906;
   DATA[2328,2] := 2.0;
   DATA[2328,3] := 2.0;
   DATA[2328,4] := 262.3366;
   DATA[2328,5] := 8.395475;
   DATA[2328,6] := 329.8898;
   DATA[2328,7] := 2.455259;
   DATA[2328,8] := 2.0;
   DATA[2328,9] := 2.0;
   DATA[2328,10] := 2.0;
   DATA[2328,11] := 19.7804;
   DATA[2328,12] := 2.210166;
   DATA[2328,13] := 814.2544;
   DATA[2328,14] := 1.0;
   DATA[2328,15] := 2.0;
   DATA[2328,16] := 1.0;
   DATA[2328,17] := 1.0;
   DATA[2328,18] := 1.0;
   DATA[2328,19] := 2.0;
   DATA[2328,20] := 148.808;
   DATA[2328,21] := 155.1653;
   DATA[2328,22] := 1.715311;
   DATA[2328,23] := 855.6268;
   DATA[2328,24] := 2.0;
   DATA[2328,25] := 2.0;
   DATA[2328,26] := 7.874135;
   DATA[2328,27] := 144.3989;
   DATA[2328,28] := 261.7278;
   DATA[2328,29] := 11.95847;
   DATA[2328,30] := 1.725455;
   DATA[2328,31] := 1.274497;
   DATA[2328,32] := 0.7353967;
   DATA[2328,33] := 0.3083624;
   DATA[2328,34] := 2.0;
   DATA[2328,35] := 249.9519;
   DATA[2328,36] := 1.730048;
   DATA[2328,37] := 188.8138;
   DATA[2328,38] := 0.000128152;
   DATA[2328,39] := 1.0;
   DATA[2328,40] := 1.0;
   DATA[2329,0] := 2.600327;
   DATA[2329,1] := 866.3083;
   DATA[2329,2] := 2.0;
   DATA[2329,3] := 2.0;
   DATA[2329,4] := 262.3366;
   DATA[2329,5] := 8.395475;
   DATA[2329,6] := 329.8898;
   DATA[2329,7] := 2.455515;
   DATA[2329,8] := 2.0;
   DATA[2329,9] := 2.0;
   DATA[2329,10] := 2.0;
   DATA[2329,11] := 19.74838;
   DATA[2329,12] := 2.210166;
   DATA[2329,13] := 814.3345;
   DATA[2329,14] := 1.0;
   DATA[2329,15] := 2.0;
   DATA[2329,16] := 1.0;
   DATA[2329,17] := 1.0;
   DATA[2329,18] := 1.0;
   DATA[2329,19] := 2.0;
   DATA[2329,20] := 148.808;
   DATA[2329,21] := 155.1653;
   DATA[2329,22] := 1.715311;
   DATA[2329,23] := 855.4345;
   DATA[2329,24] := 2.0;
   DATA[2329,25] := 2.0;
   DATA[2329,26] := 7.874135;
   DATA[2329,27] := 144.3989;
   DATA[2329,28] := 261.7278;
   DATA[2329,29] := 11.95847;
   DATA[2329,30] := 1.725455;
   DATA[2329,31] := 1.27232;
   DATA[2329,32] := 0.7353967;
   DATA[2329,33] := 0.3083624;
   DATA[2329,34] := 2.0;
   DATA[2329,35] := 250.0961;
   DATA[2329,36] := 1.730048;
   DATA[2329,37] := 188.8939;
   DATA[2329,38] := 0.000128152;
   DATA[2329,39] := 1.0;
   DATA[2329,40] := 1.0;
   DATA[2330,0] := 2.600327;
   DATA[2330,1] := 866.3083;
   DATA[2330,2] := 2.0;
   DATA[2330,3] := 2.0;
   DATA[2330,4] := 262.3366;
   DATA[2330,5] := 8.395475;
   DATA[2330,6] := 329.8898;
   DATA[2330,7] := 2.455515;
   DATA[2330,8] := 2.0;
   DATA[2330,9] := 2.0;
   DATA[2330,10] := 2.0;
   DATA[2330,11] := 19.74838;
   DATA[2330,12] := 2.210166;
   DATA[2330,13] := 814.3345;
   DATA[2330,14] := 1.0;
   DATA[2330,15] := 2.0;
   DATA[2330,16] := 1.0;
   DATA[2330,17] := 1.0;
   DATA[2330,18] := 1.0;
   DATA[2330,19] := 2.0;
   DATA[2330,20] := 148.808;
   DATA[2330,21] := 155.1653;
   DATA[2330,22] := 1.715311;
   DATA[2330,23] := 855.4345;
   DATA[2330,24] := 2.0;
   DATA[2330,25] := 2.0;
   DATA[2330,26] := 7.874135;
   DATA[2330,27] := 144.3989;
   DATA[2330,28] := 261.7278;
   DATA[2330,29] := 11.95847;
   DATA[2330,30] := 1.725455;
   DATA[2330,31] := 1.27232;
   DATA[2330,32] := 0.7353967;
   DATA[2330,33] := 0.3083624;
   DATA[2330,34] := 2.0;
   DATA[2330,35] := 250.0961;
   DATA[2330,36] := 1.730048;
   DATA[2330,37] := 188.8939;
   DATA[2330,38] := 0.000128152;
   DATA[2330,39] := 1.0;
   DATA[2330,40] := 1.0;
   DATA[2331,0] := 2.624988;
   DATA[2331,1] := 865.7589;
   DATA[2331,2] := 2.0;
   DATA[2331,3] := 2.0;
   DATA[2331,4] := 262.3366;
   DATA[2331,5] := 8.395475;
   DATA[2331,6] := 329.8898;
   DATA[2331,7] := 2.455515;
   DATA[2331,8] := 2.0;
   DATA[2331,9] := 2.0;
   DATA[2331,10] := 2.0;
   DATA[2331,11] := 19.71957;
   DATA[2331,12] := 2.210166;
   DATA[2331,13] := 813.934;
   DATA[2331,14] := 1.0;
   DATA[2331,15] := 2.0;
   DATA[2331,16] := 1.0;
   DATA[2331,17] := 1.0;
   DATA[2331,18] := 1.0;
   DATA[2331,19] := 2.0;
   DATA[2331,20] := 148.808;
   DATA[2331,21] := 155.1653;
   DATA[2331,22] := 1.717874;
   DATA[2331,23] := 855.6268;
   DATA[2331,24] := 2.0;
   DATA[2331,25] := 2.0;
   DATA[2331,26] := 7.874135;
   DATA[2331,27] := 144.3989;
   DATA[2331,28] := 261.7278;
   DATA[2331,29] := 11.95847;
   DATA[2331,30] := 1.725455;
   DATA[2331,31] := 1.28103;
   DATA[2331,32] := 0.7353967;
   DATA[2331,33] := 0.3083624;
   DATA[2331,34] := 2.0;
   DATA[2331,35] := 250.0961;
   DATA[2331,36] := 1.665972;
   DATA[2331,37] := 189.0381;
   DATA[2331,38] := 0.000128152;
   DATA[2331,39] := 1.0;
   DATA[2331,40] := 1.0;
   DATA[2332,0] := 2.652532;
   DATA[2332,1] := 865.9158;
   DATA[2332,2] := 2.0;
   DATA[2332,3] := 2.0;
   DATA[2332,4] := 262.3366;
   DATA[2332,5] := 8.395475;
   DATA[2332,6] := 329.8898;
   DATA[2332,7] := 2.453849;
   DATA[2332,8] := 2.0;
   DATA[2332,9] := 2.0;
   DATA[2332,10] := 2.0;
   DATA[2332,11] := 19.71957;
   DATA[2332,12] := 2.210166;
   DATA[2332,13] := 813.5334;
   DATA[2332,14] := 1.0;
   DATA[2332,15] := 2.0;
   DATA[2332,16] := 1.0;
   DATA[2332,17] := 1.0;
   DATA[2332,18] := 1.0;
   DATA[2332,19] := 2.0;
   DATA[2332,20] := 148.808;
   DATA[2332,21] := 155.1653;
   DATA[2332,22] := 1.717874;
   DATA[2332,23] := 855.6268;
   DATA[2332,24] := 2.0;
   DATA[2332,25] := 2.0;
   DATA[2332,26] := 7.874135;
   DATA[2332,27] := 144.3989;
   DATA[2332,28] := 261.7278;
   DATA[2332,29] := 11.95847;
   DATA[2332,30] := 1.725455;
   DATA[2332,31] := 1.281286;
   DATA[2332,32] := 0.7353967;
   DATA[2332,33] := 0.3083624;
   DATA[2332,34] := 2.0;
   DATA[2332,35] := 250.3845;
   DATA[2332,36] := 1.665972;
   DATA[2332,37] := 189.0541;
   DATA[2332,38] := 0.000128152;
   DATA[2332,39] := 1.0;
   DATA[2332,40] := 1.0;
   DATA[2333,0] := 2.658617;
   DATA[2333,1] := 865.5233;
   DATA[2333,2] := 2.0;
   DATA[2333,3] := 2.0;
   DATA[2333,4] := 262.3366;
   DATA[2333,5] := 8.398039;
   DATA[2333,6] := 329.8898;
   DATA[2333,7] := 2.453849;
   DATA[2333,8] := 2.0;
   DATA[2333,9] := 2.0;
   DATA[2333,10] := 2.0;
   DATA[2333,11] := 19.71957;
   DATA[2333,12] := 2.209269;
   DATA[2333,13] := 813.1729;
   DATA[2333,14] := 1.0;
   DATA[2333,15] := 2.0;
   DATA[2333,16] := 1.0;
   DATA[2333,17] := 1.0;
   DATA[2333,18] := 1.0;
   DATA[2333,19] := 2.0;
   DATA[2333,20] := 148.808;
   DATA[2333,21] := 155.1653;
   DATA[2333,22] := 1.717874;
   DATA[2333,23] := 855.3192;
   DATA[2333,24] := 2.0;
   DATA[2333,25] := 2.0;
   DATA[2333,26] := 7.874135;
   DATA[2333,27] := 144.3989;
   DATA[2333,28] := 261.7278;
   DATA[2333,29] := 11.95847;
   DATA[2333,30] := 1.726609;
   DATA[2333,31] := 1.291149;
   DATA[2333,32] := 0.7353967;
   DATA[2333,33] := 0.3083624;
   DATA[2333,34] := 2.0;
   DATA[2333,35] := 250.3845;
   DATA[2333,36] := 1.665972;
   DATA[2333,37] := 189.1182;
   DATA[2333,38] := 0.000128152;
   DATA[2333,39] := 1.0;
   DATA[2333,40] := 1.0;
   DATA[2334,0] := 2.658617;
   DATA[2334,1] := 865.6018;
   DATA[2334,2] := 2.0;
   DATA[2334,3] := 2.0;
   DATA[2334,4] := 262.3366;
   DATA[2334,5] := 8.398039;
   DATA[2334,6] := 329.8898;
   DATA[2334,7] := 2.453849;
   DATA[2334,8] := 2.0;
   DATA[2334,9] := 2.0;
   DATA[2334,10] := 2.0;
   DATA[2334,11] := 19.71957;
   DATA[2334,12] := 2.208628;
   DATA[2334,13] := 813.0527;
   DATA[2334,14] := 1.0;
   DATA[2334,15] := 2.0;
   DATA[2334,16] := 1.0;
   DATA[2334,17] := 1.0;
   DATA[2334,18] := 1.0;
   DATA[2334,19] := 2.0;
   DATA[2334,20] := 148.808;
   DATA[2334,21] := 155.1653;
   DATA[2334,22] := 1.717874;
   DATA[2334,23] := 855.3192;
   DATA[2334,24] := 2.0;
   DATA[2334,25] := 2.0;
   DATA[2334,26] := 7.874135;
   DATA[2334,27] := 144.3989;
   DATA[2334,28] := 261.7278;
   DATA[2334,29] := 11.95847;
   DATA[2334,30] := 1.727378;
   DATA[2334,31] := 1.291789;
   DATA[2334,32] := 0.7353967;
   DATA[2334,33] := 0.3083624;
   DATA[2334,34] := 2.0;
   DATA[2334,35] := 250.3845;
   DATA[2334,36] := 1.665972;
   DATA[2334,37] := 189.1662;
   DATA[2334,38] := 0.000128152;
   DATA[2334,39] := 1.0;
   DATA[2334,40] := 1.0;
   DATA[2335,0] := 2.638119;
   DATA[2335,1] := 865.5233;
   DATA[2335,2] := 2.0;
   DATA[2335,3] := 2.0;
   DATA[2335,4] := 262.3366;
   DATA[2335,5] := 8.398039;
   DATA[2335,6] := 329.8898;
   DATA[2335,7] := 2.453849;
   DATA[2335,8] := 2.0;
   DATA[2335,9] := 2.0;
   DATA[2335,10] := 2.0;
   DATA[2335,11] := 19.71957;
   DATA[2335,12] := 2.208628;
   DATA[2335,13] := 812.9326;
   DATA[2335,14] := 1.0;
   DATA[2335,15] := 2.0;
   DATA[2335,16] := 1.0;
   DATA[2335,17] := 1.0;
   DATA[2335,18] := 1.0;
   DATA[2335,19] := 2.0;
   DATA[2335,20] := 148.808;
   DATA[2335,21] := 155.3448;
   DATA[2335,22] := 1.718771;
   DATA[2335,23] := 855.1653;
   DATA[2335,24] := 2.0;
   DATA[2335,25] := 2.0;
   DATA[2335,26] := 7.874135;
   DATA[2335,27] := 144.3989;
   DATA[2335,28] := 261.7278;
   DATA[2335,29] := 11.95847;
   DATA[2335,30] := 1.727378;
   DATA[2335,31] := 1.291789;
   DATA[2335,32] := 0.7353967;
   DATA[2335,33] := 0.3083624;
   DATA[2335,34] := 2.0;
   DATA[2335,35] := 250.4166;
   DATA[2335,36] := 1.665972;
   DATA[2335,37] := 189.3425;
   DATA[2335,38] := 0.000128152;
   DATA[2335,39] := 1.0;
   DATA[2335,40] := 1.0;
   DATA[2336,0] := 2.626589;
   DATA[2336,1] := 865.5233;
   DATA[2336,2] := 2.0;
   DATA[2336,3] := 2.0;
   DATA[2336,4] := 262.3366;
   DATA[2336,5] := 8.398039;
   DATA[2336,6] := 329.8898;
   DATA[2336,7] := 2.45449;
   DATA[2336,8] := 2.0;
   DATA[2336,9] := 2.0;
   DATA[2336,10] := 2.0;
   DATA[2336,11] := 19.71957;
   DATA[2336,12] := 2.205682;
   DATA[2336,13] := 813.1729;
   DATA[2336,14] := 1.0;
   DATA[2336,15] := 2.0;
   DATA[2336,16] := 1.0;
   DATA[2336,17] := 1.0;
   DATA[2336,18] := 1.0;
   DATA[2336,19] := 2.0;
   DATA[2336,20] := 148.808;
   DATA[2336,21] := 155.3448;
   DATA[2336,22] := 1.721334;
   DATA[2336,23] := 855.473;
   DATA[2336,24] := 2.0;
   DATA[2336,25] := 2.0;
   DATA[2336,26] := 7.874135;
   DATA[2336,27] := 144.3989;
   DATA[2336,28] := 261.7278;
   DATA[2336,29] := 11.95847;
   DATA[2336,30] := 1.727378;
   DATA[2336,31] := 1.291789;
   DATA[2336,32] := 0.7353967;
   DATA[2336,33] := 0.3072094;
   DATA[2336,34] := 2.0;
   DATA[2336,35] := 250.4967;
   DATA[2336,36] := 1.665972;
   DATA[2336,37] := 189.3425;
   DATA[2336,38] := 0.000128152;
   DATA[2336,39] := 1.0;
   DATA[2336,40] := 1.0;
   DATA[2337,0] := 2.624988;
   DATA[2337,1] := 865.1308;
   DATA[2337,2] := 2.0;
   DATA[2337,3] := 2.0;
   DATA[2337,4] := 262.3366;
   DATA[2337,5] := 8.398039;
   DATA[2337,6] := 329.8898;
   DATA[2337,7] := 2.45449;
   DATA[2337,8] := 2.0;
   DATA[2337,9] := 2.0;
   DATA[2337,10] := 2.0;
   DATA[2337,11] := 19.74198;
   DATA[2337,12] := 2.205169;
   DATA[2337,13] := 813.5735;
   DATA[2337,14] := 1.0;
   DATA[2337,15] := 2.0;
   DATA[2337,16] := 1.0;
   DATA[2337,17] := 1.0;
   DATA[2337,18] := 1.0;
   DATA[2337,19] := 2.0;
   DATA[2337,20] := 148.808;
   DATA[2337,21] := 155.3448;
   DATA[2337,22] := 1.721334;
   DATA[2337,23] := 855.3576;
   DATA[2337,24] := 2.0;
   DATA[2337,25] := 2.0;
   DATA[2337,26] := 7.874135;
   DATA[2337,27] := 144.3989;
   DATA[2337,28] := 261.7278;
   DATA[2337,29] := 11.95847;
   DATA[2337,30] := 1.728788;
   DATA[2337,31] := 1.291789;
   DATA[2337,32] := 0.7353967;
   DATA[2337,33] := 0.3068251;
   DATA[2337,34] := 2.0;
   DATA[2337,35] := 250.4967;
   DATA[2337,36] := 1.665972;
   DATA[2337,37] := 189.3425;
   DATA[2337,38] := 0.000128152;
   DATA[2337,39] := 1.0;
   DATA[2337,40] := 1.0;
   DATA[2338,0] := 2.609615;
   DATA[2338,1] := 865.5626;
   DATA[2338,2] := 2.0;
   DATA[2338,3] := 2.0;
   DATA[2338,4] := 262.3366;
   DATA[2338,5] := 8.398039;
   DATA[2338,6] := 329.8898;
   DATA[2338,7] := 2.45449;
   DATA[2338,8] := 2.0;
   DATA[2338,9] := 2.0;
   DATA[2338,10] := 2.0;
   DATA[2338,11] := 19.74198;
   DATA[2338,12] := 2.205169;
   DATA[2338,13] := 813.5334;
   DATA[2338,14] := 1.0;
   DATA[2338,15] := 2.0;
   DATA[2338,16] := 1.0;
   DATA[2338,17] := 1.0;
   DATA[2338,18] := 1.0;
   DATA[2338,19] := 2.0;
   DATA[2338,20] := 148.808;
   DATA[2338,21] := 155.3448;
   DATA[2338,22] := 1.721334;
   DATA[2338,23] := 855.473;
   DATA[2338,24] := 2.0;
   DATA[2338,25] := 2.0;
   DATA[2338,26] := 7.874135;
   DATA[2338,27] := 144.322;
   DATA[2338,28] := 261.7278;
   DATA[2338,29] := 11.95847;
   DATA[2338,30] := 1.728788;
   DATA[2338,31] := 1.291789;
   DATA[2338,32] := 0.7353967;
   DATA[2338,33] := 0.3068251;
   DATA[2338,34] := 2.0;
   DATA[2338,35] := 250.4967;
   DATA[2338,36] := 1.665972;
   DATA[2338,37] := 189.3425;
   DATA[2338,38] := 0.000128152;
   DATA[2338,39] := 1.0;
   DATA[2338,40] := 1.0;
   DATA[2339,0] := 2.593921;
   DATA[2339,1] := 865.7589;
   DATA[2339,2] := 2.0;
   DATA[2339,3] := 2.0;
   DATA[2339,4] := 262.3366;
   DATA[2339,5] := 8.398039;
   DATA[2339,6] := 329.8898;
   DATA[2339,7] := 2.45449;
   DATA[2339,8] := 2.0;
   DATA[2339,9] := 2.0;
   DATA[2339,10] := 2.0;
   DATA[2339,11] := 19.74198;
   DATA[2339,12] := 2.20645;
   DATA[2339,13] := 813.8138;
   DATA[2339,14] := 1.0;
   DATA[2339,15] := 2.0;
   DATA[2339,16] := 1.0;
   DATA[2339,17] := 1.0;
   DATA[2339,18] := 1.0;
   DATA[2339,19] := 2.0;
   DATA[2339,20] := 148.808;
   DATA[2339,21] := 155.3448;
   DATA[2339,22] := 1.721334;
   DATA[2339,23] := 855.6268;
   DATA[2339,24] := 2.0;
   DATA[2339,25] := 2.0;
   DATA[2339,26] := 7.874135;
   DATA[2339,27] := 144.2194;
   DATA[2339,28] := 261.7278;
   DATA[2339,29] := 11.95847;
   DATA[2339,30] := 1.728788;
   DATA[2339,31] := 1.273985;
   DATA[2339,32] := 0.7353967;
   DATA[2339,33] := 0.3084905;
   DATA[2339,34] := 2.0;
   DATA[2339,35] := 250.4967;
   DATA[2339,36] := 1.665972;
   DATA[2339,37] := 189.1983;
   DATA[2339,38] := 0.000128152;
   DATA[2339,39] := 1.0;
   DATA[2339,40] := 1.0;
   DATA[2340,0] := 2.574384;
   DATA[2340,1] := 865.6018;
   DATA[2340,2] := 2.0;
   DATA[2340,3] := 2.0;
   DATA[2340,4] := 262.3366;
   DATA[2340,5] := 8.398039;
   DATA[2340,6] := 329.8898;
   DATA[2340,7] := 2.45449;
   DATA[2340,8] := 2.0;
   DATA[2340,9] := 2.0;
   DATA[2340,10] := 2.0;
   DATA[2340,11] := 19.73238;
   DATA[2340,12] := 2.20645;
   DATA[2340,13] := 813.974;
   DATA[2340,14] := 1.0;
   DATA[2340,15] := 2.0;
   DATA[2340,16] := 1.0;
   DATA[2340,17] := 1.0;
   DATA[2340,18] := 1.0;
   DATA[2340,19] := 2.0;
   DATA[2340,20] := 148.808;
   DATA[2340,21] := 155.2166;
   DATA[2340,22] := 1.720437;
   DATA[2340,23] := 855.6652;
   DATA[2340,24] := 2.0;
   DATA[2340,25] := 2.0;
   DATA[2340,26] := 7.874135;
   DATA[2340,27] := 144.2194;
   DATA[2340,28] := 261.7278;
   DATA[2340,29] := 11.95847;
   DATA[2340,30] := 1.728788;
   DATA[2340,31] := 1.271551;
   DATA[2340,32] := 0.7353967;
   DATA[2340,33] := 0.3084905;
   DATA[2340,34] := 2.0;
   DATA[2340,35] := 250.4967;
   DATA[2340,36] := 1.665972;
   DATA[2340,37] := 189.0861;
   DATA[2340,38] := 0.000128152;
   DATA[2340,39] := 1.0;
   DATA[2340,40] := 1.0;
   DATA[2341,0] := 2.562854;
   DATA[2341,1] := 865.5233;
   DATA[2341,2] := 2.0;
   DATA[2341,3] := 2.0;
   DATA[2341,4] := 262.3366;
   DATA[2341,5] := 8.398039;
   DATA[2341,6] := 329.8898;
   DATA[2341,7] := 2.455515;
   DATA[2341,8] := 2.0;
   DATA[2341,9] := 2.0;
   DATA[2341,10] := 2.0;
   DATA[2341,11] := 19.70997;
   DATA[2341,12] := 2.208244;
   DATA[2341,13] := 813.7737;
   DATA[2341,14] := 1.0;
   DATA[2341,15] := 2.0;
   DATA[2341,16] := 1.0;
   DATA[2341,17] := 1.0;
   DATA[2341,18] := 1.0;
   DATA[2341,19] := 2.0;
   DATA[2341,20] := 148.808;
   DATA[2341,21] := 155.2166;
   DATA[2341,22] := 1.719027;
   DATA[2341,23] := 856.0113;
   DATA[2341,24] := 2.0;
   DATA[2341,25] := 2.0;
   DATA[2341,26] := 7.874135;
   DATA[2341,27] := 144.2194;
   DATA[2341,28] := 261.7278;
   DATA[2341,29] := 11.95847;
   DATA[2341,30] := 1.726993;
   DATA[2341,31] := 1.270911;
   DATA[2341,32] := 0.7353967;
   DATA[2341,33] := 0.3084905;
   DATA[2341,34] := 2.0;
   DATA[2341,35] := 250.3204;
   DATA[2341,36] := 1.665972;
   DATA[2341,37] := 189.0861;
   DATA[2341,38] := 0.000128152;
   DATA[2341,39] := 1.0;
   DATA[2341,40] := 1.0;
   DATA[2342,0] := 2.542677;
   DATA[2342,1] := 865.013;
   DATA[2342,2] := 2.0;
   DATA[2342,3] := 2.0;
   DATA[2342,4] := 262.3366;
   DATA[2342,5] := 8.398039;
   DATA[2342,6] := 329.8898;
   DATA[2342,7] := 2.455515;
   DATA[2342,8] := 2.0;
   DATA[2342,9] := 2.0;
   DATA[2342,10] := 2.0;
   DATA[2342,11] := 19.70997;
   DATA[2342,12] := 2.208756;
   DATA[2342,13] := 814.0541;
   DATA[2342,14] := 1.0;
   DATA[2342,15] := 2.0;
   DATA[2342,16] := 1.0;
   DATA[2342,17] := 1.0;
   DATA[2342,18] := 1.0;
   DATA[2342,19] := 2.0;
   DATA[2342,20] := 148.808;
   DATA[2342,21] := 155.2166;
   DATA[2342,22] := 1.719027;
   DATA[2342,23] := 856.0497;
   DATA[2342,24] := 2.0;
   DATA[2342,25] := 2.0;
   DATA[2342,26] := 7.874135;
   DATA[2342,27] := 144.2194;
   DATA[2342,28] := 261.7278;
   DATA[2342,29] := 11.95847;
   DATA[2342,30] := 1.72507;
   DATA[2342,31] := 1.262329;
   DATA[2342,32] := 0.7353967;
   DATA[2342,33] := 0.3084905;
   DATA[2342,34] := 2.0;
   DATA[2342,35] := 250.3204;
   DATA[2342,36] := 1.617916;
   DATA[2342,37] := 189.0861;
   DATA[2342,38] := 0.000128152;
   DATA[2342,39] := 1.0;
   DATA[2342,40] := 1.0;
   DATA[2343,0] := 2.528264;
   DATA[2343,1] := 864.4635;
   DATA[2343,2] := 2.0;
   DATA[2343,3] := 2.0;
   DATA[2343,4] := 262.3366;
   DATA[2343,5] := 8.398039;
   DATA[2343,6] := 329.8898;
   DATA[2343,7] := 2.455515;
   DATA[2343,8] := 2.0;
   DATA[2343,9] := 2.0;
   DATA[2343,10] := 2.0;
   DATA[2343,11] := 19.74198;
   DATA[2343,12] := 2.208756;
   DATA[2343,13] := 814.4146;
   DATA[2343,14] := 1.0;
   DATA[2343,15] := 2.0;
   DATA[2343,16] := 1.0;
   DATA[2343,17] := 1.0;
   DATA[2343,18] := 1.0;
   DATA[2343,19] := 2.0;
   DATA[2343,20] := 148.808;
   DATA[2343,21] := 155.2166;
   DATA[2343,22] := 1.719027;
   DATA[2343,23] := 855.8959;
   DATA[2343,24] := 2.0;
   DATA[2343,25] := 2.0;
   DATA[2343,26] := 7.874135;
   DATA[2343,27] := 144.2194;
   DATA[2343,28] := 261.7278;
   DATA[2343,29] := 11.95847;
   DATA[2343,30] := 1.72507;
   DATA[2343,31] := 1.262457;
   DATA[2343,32] := 0.7353967;
   DATA[2343,33] := 0.3084905;
   DATA[2343,34] := 2.0;
   DATA[2343,35] := 250.2243;
   DATA[2343,36] := 1.617916;
   DATA[2343,37] := 189.0861;
   DATA[2343,38] := 0.000128152;
   DATA[2343,39] := 1.0;
   DATA[2343,40] := 1.0;
   DATA[2344,0] := 2.506485;
   DATA[2344,1] := 864.5812;
   DATA[2344,2] := 2.0;
   DATA[2344,3] := 2.0;
   DATA[2344,4] := 262.3366;
   DATA[2344,5] := 8.398039;
   DATA[2344,6] := 329.8898;
   DATA[2344,7] := 2.455515;
   DATA[2344,8] := 2.0;
   DATA[2344,9] := 2.0;
   DATA[2344,10] := 2.0;
   DATA[2344,11] := 19.74198;
   DATA[2344,12] := 2.208756;
   DATA[2344,13] := 815.1356;
   DATA[2344,14] := 1.0;
   DATA[2344,15] := 2.0;
   DATA[2344,16] := 1.0;
   DATA[2344,17] := 1.0;
   DATA[2344,18] := 1.0;
   DATA[2344,19] := 2.0;
   DATA[2344,20] := 148.808;
   DATA[2344,21] := 155.2166;
   DATA[2344,22] := 1.719027;
   DATA[2344,23] := 855.6652;
   DATA[2344,24] := 2.0;
   DATA[2344,25] := 2.0;
   DATA[2344,26] := 7.874135;
   DATA[2344,27] := 144.2194;
   DATA[2344,28] := 261.7278;
   DATA[2344,29] := 11.95847;
   DATA[2344,30] := 1.72507;
   DATA[2344,31] := 1.280389;
   DATA[2344,32] := 0.7353967;
   DATA[2344,33] := 0.3084905;
   DATA[2344,34] := 2.0;
   DATA[2344,35] := 250.2243;
   DATA[2344,36] := 1.617916;
   DATA[2344,37] := 189.0861;
   DATA[2344,38] := 0.000128152;
   DATA[2344,39] := 1.0;
   DATA[2344,40] := 1.0;
   DATA[2345,0] := 2.496877;
   DATA[2345,1] := 864.385;
   DATA[2345,2] := 2.0;
   DATA[2345,3] := 2.0;
   DATA[2345,4] := 262.3366;
   DATA[2345,5] := 8.398039;
   DATA[2345,6] := 329.8898;
   DATA[2345,7] := 2.455515;
   DATA[2345,8] := 2.0;
   DATA[2345,9] := 2.0;
   DATA[2345,10] := 2.0;
   DATA[2345,11] := 19.67796;
   DATA[2345,12] := 2.209909;
   DATA[2345,13] := 815.8165;
   DATA[2345,14] := 1.0;
   DATA[2345,15] := 2.0;
   DATA[2345,16] := 1.0;
   DATA[2345,17] := 1.0;
   DATA[2345,18] := 1.0;
   DATA[2345,19] := 2.0;
   DATA[2345,20] := 148.808;
   DATA[2345,21] := 155.2166;
   DATA[2345,22] := 1.719027;
   DATA[2345,23] := 855.8575;
   DATA[2345,24] := 2.0;
   DATA[2345,25] := 2.0;
   DATA[2345,26] := 7.874135;
   DATA[2345,27] := 144.2194;
   DATA[2345,28] := 261.7278;
   DATA[2345,29] := 11.95847;
   DATA[2345,30] := 1.72507;
   DATA[2345,31] := 1.27834;
   DATA[2345,32] := 0.7353967;
   DATA[2345,33] := 0.3084905;
   DATA[2345,34] := 2.0;
   DATA[2345,35] := 250.2243;
   DATA[2345,36] := 1.617916;
   DATA[2345,37] := 189.0861;
   DATA[2345,38] := 0.000128152;
   DATA[2345,39] := 1.0;
   DATA[2345,40] := 1.0;
   DATA[2346,0] := 2.47638;
   DATA[2346,1] := 864.542;
   DATA[2346,2] := 2.0;
   DATA[2346,3] := 2.0;
   DATA[2346,4] := 262.3366;
   DATA[2346,5] := 8.398039;
   DATA[2346,6] := 329.8898;
   DATA[2346,7] := 2.453209;
   DATA[2346,8] := 2.0;
   DATA[2346,9] := 2.0;
   DATA[2346,10] := 2.0;
   DATA[2346,11] := 19.67796;
   DATA[2346,12] := 2.21055;
   DATA[2346,13] := 816.3773;
   DATA[2346,14] := 1.0;
   DATA[2346,15] := 2.0;
   DATA[2346,16] := 1.0;
   DATA[2346,17] := 1.0;
   DATA[2346,18] := 1.0;
   DATA[2346,19] := 2.0;
   DATA[2346,20] := 148.808;
   DATA[2346,21] := 155.2166;
   DATA[2346,22] := 1.719027;
   DATA[2346,23] := 855.7421;
   DATA[2346,24] := 2.0;
   DATA[2346,25] := 2.0;
   DATA[2346,26] := 7.874135;
   DATA[2346,27] := 144.2194;
   DATA[2346,28] := 261.7278;
   DATA[2346,29] := 11.95847;
   DATA[2346,30] := 1.72507;
   DATA[2346,31] := 1.262329;
   DATA[2346,32] := 0.7353967;
   DATA[2346,33] := 0.3084905;
   DATA[2346,34] := 2.0;
   DATA[2346,35] := 250.2243;
   DATA[2346,36] := 1.617916;
   DATA[2346,37] := 189.006;
   DATA[2346,38] := 0.000128152;
   DATA[2346,39] := 1.0;
   DATA[2346,40] := 1.0;
   DATA[2347,0] := 2.464849;
   DATA[2347,1] := 864.6205;
   DATA[2347,2] := 2.0;
   DATA[2347,3] := 2.0;
   DATA[2347,4] := 262.3366;
   DATA[2347,5] := 8.398039;
   DATA[2347,6] := 329.8898;
   DATA[2347,7] := 2.453209;
   DATA[2347,8] := 2.0;
   DATA[2347,9] := 2.0;
   DATA[2347,10] := 2.0;
   DATA[2347,11] := 19.73558;
   DATA[2347,12] := 2.21055;
   DATA[2347,13] := 816.8178;
   DATA[2347,14] := 1.0;
   DATA[2347,15] := 2.0;
   DATA[2347,16] := 1.0;
   DATA[2347,17] := 1.0;
   DATA[2347,18] := 1.0;
   DATA[2347,19] := 2.0;
   DATA[2347,20] := 148.808;
   DATA[2347,21] := 155.2166;
   DATA[2347,22] := 1.719027;
   DATA[2347,23] := 855.8959;
   DATA[2347,24] := 2.0;
   DATA[2347,25] := 2.0;
   DATA[2347,26] := 7.874135;
   DATA[2347,27] := 144.2194;
   DATA[2347,28] := 261.7278;
   DATA[2347,29] := 11.95847;
   DATA[2347,30] := 1.72507;
   DATA[2347,31] := 1.267452;
   DATA[2347,32] := 0.7353967;
   DATA[2347,33] := 0.3084905;
   DATA[2347,34] := 2.0;
   DATA[2347,35] := 250.2243;
   DATA[2347,36] := 1.617916;
   DATA[2347,37] := 188.9259;
   DATA[2347,38] := 0.000128152;
   DATA[2347,39] := 1.0;
   DATA[2347,40] := 1.0;
   DATA[2348,0] := 2.449156;
   DATA[2348,1] := 864.4635;
   DATA[2348,2] := 2.0;
   DATA[2348,3] := 2.0;
   DATA[2348,4] := 262.3366;
   DATA[2348,5] := 8.398039;
   DATA[2348,6] := 329.8898;
   DATA[2348,7] := 2.453209;
   DATA[2348,8] := 2.0;
   DATA[2348,9] := 2.0;
   DATA[2348,10] := 2.0;
   DATA[2348,11] := 19.74198;
   DATA[2348,12] := 2.21055;
   DATA[2348,13] := 817.1382;
   DATA[2348,14] := 1.0;
   DATA[2348,15] := 2.0;
   DATA[2348,16] := 1.0;
   DATA[2348,17] := 1.0;
   DATA[2348,18] := 1.0;
   DATA[2348,19] := 2.0;
   DATA[2348,20] := 148.808;
   DATA[2348,21] := 155.2166;
   DATA[2348,22] := 1.716208;
   DATA[2348,23] := 856.242;
   DATA[2348,24] := 2.0;
   DATA[2348,25] := 2.0;
   DATA[2348,26] := 7.874135;
   DATA[2348,27] := 144.2194;
   DATA[2348,28] := 261.7278;
   DATA[2348,29] := 11.95847;
   DATA[2348,30] := 1.723661;
   DATA[2348,31] := 1.26758;
   DATA[2348,32] := 0.7353967;
   DATA[2348,33] := 0.3084905;
   DATA[2348,34] := 2.0;
   DATA[2348,35] := 250.016;
   DATA[2348,36] := 1.617916;
   DATA[2348,37] := 188.8458;
   DATA[2348,38] := 0.000128152;
   DATA[2348,39] := 1.0;
   DATA[2348,40] := 1.0;
   DATA[2349,0] := 2.437946;
   DATA[2349,1] := 864.856;
   DATA[2349,2] := 2.0;
   DATA[2349,3] := 2.0;
   DATA[2349,4] := 262.3366;
   DATA[2349,5] := 8.398039;
   DATA[2349,6] := 329.8898;
   DATA[2349,7] := 2.455003;
   DATA[2349,8] := 2.0;
   DATA[2349,9] := 2.0;
   DATA[2349,10] := 2.0;
   DATA[2349,11] := 19.74198;
   DATA[2349,12] := 2.21055;
   DATA[2349,13] := 817.3786;
   DATA[2349,14] := 1.0;
   DATA[2349,15] := 2.0;
   DATA[2349,16] := 1.0;
   DATA[2349,17] := 1.0;
   DATA[2349,18] := 1.0;
   DATA[2349,19] := 2.0;
   DATA[2349,20] := 148.808;
   DATA[2349,21] := 155.2166;
   DATA[2349,22] := 1.716208;
   DATA[2349,23] := 855.7037;
   DATA[2349,24] := 2.0;
   DATA[2349,25] := 2.0;
   DATA[2349,26] := 7.874135;
   DATA[2349,27] := 144.2194;
   DATA[2349,28] := 261.7278;
   DATA[2349,29] := 11.95847;
   DATA[2349,30] := 1.723404;
   DATA[2349,31] := 1.272832;
   DATA[2349,32] := 0.7353967;
   DATA[2349,33] := 0.3084905;
   DATA[2349,34] := 2.0;
   DATA[2349,35] := 250.016;
   DATA[2349,36] := 1.617916;
   DATA[2349,37] := 188.7977;
   DATA[2349,38] := 0.000128152;
   DATA[2349,39] := 1.0;
   DATA[2349,40] := 1.0;
   DATA[2350,0] := 2.43058;
   DATA[2350,1] := 864.8168;
   DATA[2350,2] := 2.0;
   DATA[2350,3] := 2.0;
   DATA[2350,4] := 262.3366;
   DATA[2350,5] := 8.398039;
   DATA[2350,6] := 329.8898;
   DATA[2350,7] := 2.455643;
   DATA[2350,8] := 2.0;
   DATA[2350,9] := 2.0;
   DATA[2350,10] := 2.0;
   DATA[2350,11] := 19.74198;
   DATA[2350,12] := 2.209525;
   DATA[2350,13] := 817.5388;
   DATA[2350,14] := 1.0;
   DATA[2350,15] := 2.0;
   DATA[2350,16] := 1.0;
   DATA[2350,17] := 1.0;
   DATA[2350,18] := 1.0;
   DATA[2350,19] := 2.0;
   DATA[2350,20] := 148.808;
   DATA[2350,21] := 155.2166;
   DATA[2350,22] := 1.715183;
   DATA[2350,23] := 856.0497;
   DATA[2350,24] := 2.0;
   DATA[2350,25] := 2.0;
   DATA[2350,26] := 7.874135;
   DATA[2350,27] := 144.2194;
   DATA[2350,28] := 261.7278;
   DATA[2350,29] := 11.95847;
   DATA[2350,30] := 1.723404;
   DATA[2350,31] := 1.293711;
   DATA[2350,32] := 0.7353967;
   DATA[2350,33] := 0.3084905;
   DATA[2350,34] := 2.0;
   DATA[2350,35] := 250.016;
   DATA[2350,36] := 1.649953;
   DATA[2350,37] := 188.7977;
   DATA[2350,38] := 0.000128152;
   DATA[2350,39] := 1.0;
   DATA[2350,40] := 1.0;
   DATA[2351,0] := 2.428979;
   DATA[2351,1] := 864.856;
   DATA[2351,2] := 2.0;
   DATA[2351,3] := 2.0;
   DATA[2351,4] := 262.3366;
   DATA[2351,5] := 8.398039;
   DATA[2351,6] := 329.8898;
   DATA[2351,7] := 2.455643;
   DATA[2351,8] := 2.0;
   DATA[2351,9] := 2.0;
   DATA[2351,10] := 2.0;
   DATA[2351,11] := 19.74198;
   DATA[2351,12] := 2.209525;
   DATA[2351,13] := 817.0181;
   DATA[2351,14] := 1.0;
   DATA[2351,15] := 2.0;
   DATA[2351,16] := 1.0;
   DATA[2351,17] := 1.0;
   DATA[2351,18] := 1.0;
   DATA[2351,19] := 2.0;
   DATA[2351,20] := 148.808;
   DATA[2351,21] := 155.2166;
   DATA[2351,22] := 1.714029;
   DATA[2351,23] := 856.3189;
   DATA[2351,24] := 2.0;
   DATA[2351,25] := 2.0;
   DATA[2351,26] := 7.874135;
   DATA[2351,27] := 144.2194;
   DATA[2351,28] := 261.7278;
   DATA[2351,29] := 11.95847;
   DATA[2351,30] := 1.723404;
   DATA[2351,31] := 1.294607;
   DATA[2351,32] := 0.7353967;
   DATA[2351,33] := 0.3084905;
   DATA[2351,34] := 2.0;
   DATA[2351,35] := 250.016;
   DATA[2351,36] := 1.649953;
   DATA[2351,37] := 188.7977;
   DATA[2351,38] := 0.000128152;
   DATA[2351,39] := 1.0;
   DATA[2351,40] := 1.0;
   DATA[2352,0] := 2.428979;
   DATA[2352,1] := 865.2093;
   DATA[2352,2] := 2.0;
   DATA[2352,3] := 2.0;
   DATA[2352,4] := 262.3366;
   DATA[2352,5] := 8.398039;
   DATA[2352,6] := 329.8898;
   DATA[2352,7] := 2.455643;
   DATA[2352,8] := 2.0;
   DATA[2352,9] := 2.0;
   DATA[2352,10] := 2.0;
   DATA[2352,11] := 19.74198;
   DATA[2352,12] := 2.211575;
   DATA[2352,13] := 817.6589;
   DATA[2352,14] := 1.0;
   DATA[2352,15] := 2.0;
   DATA[2352,16] := 1.0;
   DATA[2352,17] := 1.0;
   DATA[2352,18] := 1.0;
   DATA[2352,19] := 2.0;
   DATA[2352,20] := 148.808;
   DATA[2352,21] := 155.2166;
   DATA[2352,22] := 1.712876;
   DATA[2352,23] := 856.2805;
   DATA[2352,24] := 2.0;
   DATA[2352,25] := 2.0;
   DATA[2352,26] := 7.874135;
   DATA[2352,27] := 144.2194;
   DATA[2352,28] := 261.7278;
   DATA[2352,29] := 11.95847;
   DATA[2352,30] := 1.72443;
   DATA[2352,31] := 1.299603;
   DATA[2352,32] := 0.7353967;
   DATA[2352,33] := 0.3084905;
   DATA[2352,34] := 2.0;
   DATA[2352,35] := 250.1122;
   DATA[2352,36] := 1.649953;
   DATA[2352,37] := 188.9259;
   DATA[2352,38] := 0.000128152;
   DATA[2352,39] := 1.0;
   DATA[2352,40] := 1.0;
   DATA[2353,0] := 2.478301;
   DATA[2353,1] := 865.4056;
   DATA[2353,2] := 2.0;
   DATA[2353,3] := 2.0;
   DATA[2353,4] := 262.3366;
   DATA[2353,5] := 8.398039;
   DATA[2353,6] := 329.8898;
   DATA[2353,7] := 2.455643;
   DATA[2353,8] := 2.0;
   DATA[2353,9] := 2.0;
   DATA[2353,10] := 2.0;
   DATA[2353,11] := 19.74198;
   DATA[2353,12] := 2.211575;
   DATA[2353,13] := 818.0595;
   DATA[2353,14] := 1.0;
   DATA[2353,15] := 2.0;
   DATA[2353,16] := 1.0;
   DATA[2353,17] := 1.0;
   DATA[2353,18] := 1.0;
   DATA[2353,19] := 2.0;
   DATA[2353,20] := 148.808;
   DATA[2353,21] := 155.2166;
   DATA[2353,22] := 1.712876;
   DATA[2353,23] := 856.2805;
   DATA[2353,24] := 2.0;
   DATA[2353,25] := 2.0;
   DATA[2353,26] := 7.874135;
   DATA[2353,27] := 144.2194;
   DATA[2353,28] := 261.7278;
   DATA[2353,29] := 11.95847;
   DATA[2353,30] := 1.725455;
   DATA[2353,31] := 1.302037;
   DATA[2353,32] := 0.7353967;
   DATA[2353,33] := 0.3084905;
   DATA[2353,34] := 2.0;
   DATA[2353,35] := 250.1923;
   DATA[2353,36] := 1.649953;
   DATA[2353,37] := 188.958;
   DATA[2353,38] := 0.000128152;
   DATA[2353,39] := 1.0;
   DATA[2353,40] := 1.0;
   DATA[2354,0] := 2.524741;
   DATA[2354,1] := 865.4841;
   DATA[2354,2] := 2.0;
   DATA[2354,3] := 2.0;
   DATA[2354,4] := 262.3366;
   DATA[2354,5] := 8.398039;
   DATA[2354,6] := 329.8898;
   DATA[2354,7] := 2.455643;
   DATA[2354,8] := 2.0;
   DATA[2354,9] := 2.0;
   DATA[2354,10] := 2.0;
   DATA[2354,11] := 19.71957;
   DATA[2354,12] := 2.211575;
   DATA[2354,13] := 818.1396;
   DATA[2354,14] := 1.0;
   DATA[2354,15] := 2.0;
   DATA[2354,16] := 1.0;
   DATA[2354,17] := 1.0;
   DATA[2354,18] := 1.0;
   DATA[2354,19] := 2.0;
   DATA[2354,20] := 148.808;
   DATA[2354,21] := 155.2166;
   DATA[2354,22] := 1.712876;
   DATA[2354,23] := 856.0882;
   DATA[2354,24] := 2.0;
   DATA[2354,25] := 2.0;
   DATA[2354,26] := 7.874135;
   DATA[2354,27] := 144.2194;
   DATA[2354,28] := 261.7278;
   DATA[2354,29] := 11.95847;
   DATA[2354,30] := 1.726865;
   DATA[2354,31] := 1.294992;
   DATA[2354,32] := 0.7353967;
   DATA[2354,33] := 0.3084905;
   DATA[2354,34] := 2.0;
   DATA[2354,35] := 250.1923;
   DATA[2354,36] := 1.649953;
   DATA[2354,37] := 188.958;
   DATA[2354,38] := 0.000128152;
   DATA[2354,39] := 1.0;
   DATA[2354,40] := 1.0;
   DATA[2355,0] := 2.561253;
   DATA[2355,1] := 865.7589;
   DATA[2355,2] := 2.0;
   DATA[2355,3] := 2.0;
   DATA[2355,4] := 262.3366;
   DATA[2355,5] := 8.398039;
   DATA[2355,6] := 329.8898;
   DATA[2355,7] := 2.456412;
   DATA[2355,8] := 2.0;
   DATA[2355,9] := 2.0;
   DATA[2355,10] := 2.0;
   DATA[2355,11] := 19.67155;
   DATA[2355,12] := 2.210166;
   DATA[2355,13] := 818.46;
   DATA[2355,14] := 1.0;
   DATA[2355,15] := 2.0;
   DATA[2355,16] := 1.0;
   DATA[2355,17] := 1.0;
   DATA[2355,18] := 1.0;
   DATA[2355,19] := 2.0;
   DATA[2355,20] := 148.808;
   DATA[2355,21] := 155.2166;
   DATA[2355,22] := 1.717361;
   DATA[2355,23] := 856.665;
   DATA[2355,24] := 2.0;
   DATA[2355,25] := 2.0;
   DATA[2355,26] := 7.874135;
   DATA[2355,27] := 144.2194;
   DATA[2355,28] := 261.7278;
   DATA[2355,29] := 11.95847;
   DATA[2355,30] := 1.728659;
   DATA[2355,31] := 1.291789;
   DATA[2355,32] := 0.7353967;
   DATA[2355,33] := 0.3084905;
   DATA[2355,34] := 2.0;
   DATA[2355,35] := 250.3044;
   DATA[2355,36] := 1.649953;
   DATA[2355,37] := 189.006;
   DATA[2355,38] := 0.000128152;
   DATA[2355,39] := 1.0;
   DATA[2355,40] := 1.0;
   DATA[2356,0] := 2.601287;
   DATA[2356,1] := 865.9943;
   DATA[2356,2] := 2.0;
   DATA[2356,3] := 2.0;
   DATA[2356,4] := 262.3366;
   DATA[2356,5] := 8.398039;
   DATA[2356,6] := 329.8898;
   DATA[2356,7] := 2.456412;
   DATA[2356,8] := 2.0;
   DATA[2356,9] := 2.0;
   DATA[2356,10] := 2.0;
   DATA[2356,11] := 19.67155;
   DATA[2356,12] := 2.210166;
   DATA[2356,13] := 818.5802;
   DATA[2356,14] := 1.0;
   DATA[2356,15] := 2.0;
   DATA[2356,16] := 1.0;
   DATA[2356,17] := 1.0;
   DATA[2356,18] := 1.0;
   DATA[2356,19] := 2.0;
   DATA[2356,20] := 148.808;
   DATA[2356,21] := 155.2166;
   DATA[2356,22] := 1.717361;
   DATA[2356,23] := 857.2802;
   DATA[2356,24] := 2.0;
   DATA[2356,25] := 2.0;
   DATA[2356,26] := 7.874135;
   DATA[2356,27] := 144.2194;
   DATA[2356,28] := 261.7278;
   DATA[2356,29] := 12.11228;
   DATA[2356,30] := 1.728659;
   DATA[2356,31] := 1.291789;
   DATA[2356,32] := 0.7353967;
   DATA[2356,33] := 0.3084905;
   DATA[2356,34] := 2.0;
   DATA[2356,35] := 250.3044;
   DATA[2356,36] := 1.649953;
   DATA[2356,37] := 189.2143;
   DATA[2356,38] := 0.000128152;
   DATA[2356,39] := 1.0;
   DATA[2356,40] := 1.0;
   DATA[2357,0] := 2.632354;
   DATA[2357,1] := 866.5831;
   DATA[2357,2] := 2.0;
   DATA[2357,3] := 2.0;
   DATA[2357,4] := 262.3366;
   DATA[2357,5] := 8.398039;
   DATA[2357,6] := 329.8898;
   DATA[2357,7] := 2.456412;
   DATA[2357,8] := 2.0;
   DATA[2357,9] := 2.0;
   DATA[2357,10] := 2.0;
   DATA[2357,11] := 19.67155;
   DATA[2357,12] := 2.210166;
   DATA[2357,13] := 818.42;
   DATA[2357,14] := 1.0;
   DATA[2357,15] := 2.0;
   DATA[2357,16] := 1.0;
   DATA[2357,17] := 1.0;
   DATA[2357,18] := 1.0;
   DATA[2357,19] := 2.0;
   DATA[2357,20] := 148.808;
   DATA[2357,21] := 155.2166;
   DATA[2357,22] := 1.717489;
   DATA[2357,23] := 857.4725;
   DATA[2357,24] := 2.0;
   DATA[2357,25] := 2.0;
   DATA[2357,26] := 7.874135;
   DATA[2357,27] := 144.2194;
   DATA[2357,28] := 261.7278;
   DATA[2357,29] := 12.11228;
   DATA[2357,30] := 1.728659;
   DATA[2357,31] := 1.273857;
   DATA[2357,32] := 0.7353967;
   DATA[2357,33] := 0.3084905;
   DATA[2357,34] := 2.0;
   DATA[2357,35] := 250.3044;
   DATA[2357,36] := 1.649953;
   DATA[2357,37] := 189.2143;
   DATA[2357,38] := 0.000128152;
   DATA[2357,39] := 1.0;
   DATA[2357,40] := 1.0;
   DATA[2358,0] := 2.651251;
   DATA[2358,1] := 866.7402;
   DATA[2358,2] := 2.0;
   DATA[2358,3] := 2.0;
   DATA[2358,4] := 262.3366;
   DATA[2358,5] := 8.398039;
   DATA[2358,6] := 329.8898;
   DATA[2358,7] := 2.456412;
   DATA[2358,8] := 2.0;
   DATA[2358,9] := 2.0;
   DATA[2358,10] := 2.0;
   DATA[2358,11] := 19.66195;
   DATA[2358,12] := 2.210166;
   DATA[2358,13] := 818.7404;
   DATA[2358,14] := 1.0;
   DATA[2358,15] := 2.0;
   DATA[2358,16] := 1.0;
   DATA[2358,17] := 1.0;
   DATA[2358,18] := 1.0;
   DATA[2358,19] := 2.0;
   DATA[2358,20] := 148.808;
   DATA[2358,21] := 155.2166;
   DATA[2358,22] := 1.717489;
   DATA[2358,23] := 857.5493;
   DATA[2358,24] := 2.0;
   DATA[2358,25] := 2.0;
   DATA[2358,26] := 7.874135;
   DATA[2358,27] := 144.2194;
   DATA[2358,28] := 261.7278;
   DATA[2358,29] := 12.11228;
   DATA[2358,30] := 1.728659;
   DATA[2358,31] := 1.27834;
   DATA[2358,32] := 0.7353967;
   DATA[2358,33] := 0.3084905;
   DATA[2358,34] := 2.0;
   DATA[2358,35] := 250.3044;
   DATA[2358,36] := 1.649953;
   DATA[2358,37] := 189.0541;
   DATA[2358,38] := 0.000128152;
   DATA[2358,39] := 1.0;
   DATA[2358,40] := 1.0;
   DATA[2359,0] := 2.655414;
   DATA[2359,1] := 866.8972;
   DATA[2359,2] := 2.0;
   DATA[2359,3] := 2.0;
   DATA[2359,4] := 262.3366;
   DATA[2359,5] := 8.398039;
   DATA[2359,6] := 329.8898;
   DATA[2359,7] := 2.456412;
   DATA[2359,8] := 2.0;
   DATA[2359,9] := 2.0;
   DATA[2359,10] := 2.0;
   DATA[2359,11] := 19.66195;
   DATA[2359,12] := 2.210166;
   DATA[2359,13] := 818.3799;
   DATA[2359,14] := 1.0;
   DATA[2359,15] := 2.0;
   DATA[2359,16] := 1.0;
   DATA[2359,17] := 1.0;
   DATA[2359,18] := 1.0;
   DATA[2359,19] := 2.0;
   DATA[2359,20] := 148.808;
   DATA[2359,21] := 155.2166;
   DATA[2359,22] := 1.719027;
   DATA[2359,23] := 857.8569;
   DATA[2359,24] := 2.0;
   DATA[2359,25] := 2.0;
   DATA[2359,26] := 7.874135;
   DATA[2359,27] := 144.2194;
   DATA[2359,28] := 261.7278;
   DATA[2359,29] := 12.11228;
   DATA[2359,30] := 1.728659;
   DATA[2359,31] := 1.282311;
   DATA[2359,32] := 0.7353967;
   DATA[2359,33] := 0.3084905;
   DATA[2359,34] := 2.0;
   DATA[2359,35] := 250.2724;
   DATA[2359,36] := 1.649953;
   DATA[2359,37] := 189.0541;
   DATA[2359,38] := 0.000128152;
   DATA[2359,39] := 1.0;
   DATA[2359,40] := 1.0;
   DATA[2360,0] := 2.657976;
   DATA[2360,1] := 866.8579;
   DATA[2360,2] := 2.0;
   DATA[2360,3] := 2.0;
   DATA[2360,4] := 262.3366;
   DATA[2360,5] := 8.396437;
   DATA[2360,6] := 329.8898;
   DATA[2360,7] := 2.454362;
   DATA[2360,8] := 2.0;
   DATA[2360,9] := 2.0;
   DATA[2360,10] := 2.0;
   DATA[2360,11] := 19.73878;
   DATA[2360,12] := 2.210166;
   DATA[2360,13] := 818.6202;
   DATA[2360,14] := 1.0;
   DATA[2360,15] := 2.0;
   DATA[2360,16] := 1.0;
   DATA[2360,17] := 1.0;
   DATA[2360,18] := 1.0;
   DATA[2360,19] := 2.0;
   DATA[2360,20] := 148.808;
   DATA[2360,21] := 155.2166;
   DATA[2360,22] := 1.719027;
   DATA[2360,23] := 858.1646;
   DATA[2360,24] := 2.0;
   DATA[2360,25] := 2.0;
   DATA[2360,26] := 7.874135;
   DATA[2360,27] := 144.2194;
   DATA[2360,28] := 261.7278;
   DATA[2360,29] := 12.11228;
   DATA[2360,30] := 1.728659;
   DATA[2360,31] := 1.276034;
   DATA[2360,32] := 0.7353967;
   DATA[2360,33] := 0.3084905;
   DATA[2360,34] := 2.0;
   DATA[2360,35] := 250.1762;
   DATA[2360,36] := 1.649953;
   DATA[2360,37] := 189.0541;
   DATA[2360,38] := 0.000128152;
   DATA[2360,39] := 1.0;
   DATA[2360,40] := 1.0;
   DATA[2361,0] := 2.638119;
   DATA[2361,1] := 866.9364;
   DATA[2361,2] := 2.0;
   DATA[2361,3] := 2.0;
   DATA[2361,4] := 262.3366;
   DATA[2361,5] := 8.393232;
   DATA[2361,6] := 329.8898;
   DATA[2361,7] := 2.453593;
   DATA[2361,8] := 2.0;
   DATA[2361,9] := 2.0;
   DATA[2361,10] := 2.0;
   DATA[2361,11] := 19.73878;
   DATA[2361,12] := 2.208756;
   DATA[2361,13] := 818.2197;
   DATA[2361,14] := 1.0;
   DATA[2361,15] := 2.0;
   DATA[2361,16] := 1.0;
   DATA[2361,17] := 1.0;
   DATA[2361,18] := 1.0;
   DATA[2361,19] := 2.0;
   DATA[2361,20] := 148.808;
   DATA[2361,21] := 155.2166;
   DATA[2361,22] := 1.719027;
   DATA[2361,23] := 858.0492;
   DATA[2361,24] := 2.0;
   DATA[2361,25] := 2.0;
   DATA[2361,26] := 7.874135;
   DATA[2361,27] := 144.2194;
   DATA[2361,28] := 261.7278;
   DATA[2361,29] := 12.11228;
   DATA[2361,30] := 1.72725;
   DATA[2361,31] := 1.277699;
   DATA[2361,32] := 0.7353967;
   DATA[2361,33] := 0.3084905;
   DATA[2361,34] := 2.0;
   DATA[2361,35] := 250.1762;
   DATA[2361,36] := 1.649953;
   DATA[2361,37] := 189.0541;
   DATA[2361,38] := 0.000128152;
   DATA[2361,39] := 1.0;
   DATA[2361,40] := 1.0;
   DATA[2362,0] := 2.629792;
   DATA[2362,1] := 866.8972;
   DATA[2362,2] := 2.0;
   DATA[2362,3] := 2.0;
   DATA[2362,4] := 262.3366;
   DATA[2362,5] := 8.393232;
   DATA[2362,6] := 329.8898;
   DATA[2362,7] := 2.453593;
   DATA[2362,8] := 2.0;
   DATA[2362,9] := 2.0;
   DATA[2362,10] := 2.0;
   DATA[2362,11] := 19.73878;
   DATA[2362,12] := 2.208756;
   DATA[2362,13] := 818.3799;
   DATA[2362,14] := 1.0;
   DATA[2362,15] := 2.0;
   DATA[2362,16] := 1.0;
   DATA[2362,17] := 1.0;
   DATA[2362,18] := 1.0;
   DATA[2362,19] := 2.0;
   DATA[2362,20] := 148.808;
   DATA[2362,21] := 155.2166;
   DATA[2362,22] := 1.719027;
   DATA[2362,23] := 858.7029;
   DATA[2362,24] := 2.0;
   DATA[2362,25] := 2.0;
   DATA[2362,26] := 7.874135;
   DATA[2362,27] := 144.2194;
   DATA[2362,28] := 261.7278;
   DATA[2362,29] := 12.11228;
   DATA[2362,30] := 1.725327;
   DATA[2362,31] := 1.272192;
   DATA[2362,32] := 0.7353967;
   DATA[2362,33] := 0.3084905;
   DATA[2362,34] := 2.0;
   DATA[2362,35] := 250.1762;
   DATA[2362,36] := 1.649953;
   DATA[2362,37] := 189.0541;
   DATA[2362,38] := 0.000128152;
   DATA[2362,39] := 1.0;
   DATA[2362,40] := 1.0;
   DATA[2363,0] := 2.624347;
   DATA[2363,1] := 866.8972;
   DATA[2363,2] := 2.0;
   DATA[2363,3] := 2.0;
   DATA[2363,4] := 262.3366;
   DATA[2363,5] := 8.393232;
   DATA[2363,6] := 329.8898;
   DATA[2363,7] := 2.451799;
   DATA[2363,8] := 2.0;
   DATA[2363,9] := 2.0;
   DATA[2363,10] := 2.0;
   DATA[2363,11] := 19.73878;
   DATA[2363,12] := 2.208756;
   DATA[2363,13] := 818.2598;
   DATA[2363,14] := 1.0;
   DATA[2363,15] := 2.0;
   DATA[2363,16] := 1.0;
   DATA[2363,17] := 1.0;
   DATA[2363,18] := 1.0;
   DATA[2363,19] := 2.0;
   DATA[2363,20] := 148.808;
   DATA[2363,21] := 155.2166;
   DATA[2363,22] := 1.717874;
   DATA[2363,23] := 859.3181;
   DATA[2363,24] := 2.0;
   DATA[2363,25] := 2.0;
   DATA[2363,26] := 7.874135;
   DATA[2363,27] := 144.2194;
   DATA[2363,28] := 261.7278;
   DATA[2363,29] := 12.11228;
   DATA[2363,30] := 1.72443;
   DATA[2363,31] := 1.261944;
   DATA[2363,32] := 0.7353967;
   DATA[2363,33] := 0.3084905;
   DATA[2363,34] := 2.0;
   DATA[2363,35] := 250.1762;
   DATA[2363,36] := 1.649953;
   DATA[2363,37] := 189.0541;
   DATA[2363,38] := 0.000128152;
   DATA[2363,39] := 1.0;
   DATA[2363,40] := 1.0;
   DATA[2364,0] := 2.618582;
   DATA[2364,1] := 866.7794;
   DATA[2364,2] := 2.0;
   DATA[2364,3] := 2.0;
   DATA[2364,4] := 262.3366;
   DATA[2364,5] := 8.393232;
   DATA[2364,6] := 329.8898;
   DATA[2364,7] := 2.451799;
   DATA[2364,8] := 2.0;
   DATA[2364,9] := 2.0;
   DATA[2364,10] := 2.0;
   DATA[2364,11] := 19.70037;
   DATA[2364,12] := 2.208756;
   DATA[2364,13] := 818.2197;
   DATA[2364,14] := 1.0;
   DATA[2364,15] := 2.0;
   DATA[2364,16] := 1.0;
   DATA[2364,17] := 1.0;
   DATA[2364,18] := 1.0;
   DATA[2364,19] := 2.0;
   DATA[2364,20] := 148.808;
   DATA[2364,21] := 155.2166;
   DATA[2364,22] := 1.717874;
   DATA[2364,23] := 858.9336;
   DATA[2364,24] := 2.0;
   DATA[2364,25] := 2.0;
   DATA[2364,26] := 7.874135;
   DATA[2364,27] := 144.2194;
   DATA[2364,28] := 261.7278;
   DATA[2364,29] := 12.11228;
   DATA[2364,30] := 1.72443;
   DATA[2364,31] := 1.269117;
   DATA[2364,32] := 0.7353967;
   DATA[2364,33] := 0.3070813;
   DATA[2364,34] := 2.0;
   DATA[2364,35] := 250.1762;
   DATA[2364,36] := 1.762086;
   DATA[2364,37] := 189.0381;
   DATA[2364,38] := 0.000128152;
   DATA[2364,39] := 1.0;
   DATA[2364,40] := 1.0;
   DATA[2365,0] := 2.596483;
   DATA[2365,1] := 867.0542;
   DATA[2365,2] := 2.0;
   DATA[2365,3] := 2.0;
   DATA[2365,4] := 262.3366;
   DATA[2365,5] := 8.393232;
   DATA[2365,6] := 329.8898;
   DATA[2365,7] := 2.452568;
   DATA[2365,8] := 2.0;
   DATA[2365,9] := 2.0;
   DATA[2365,10] := 2.0;
   DATA[2365,11] := 19.68756;
   DATA[2365,12] := 2.209909;
   DATA[2365,13] := 817.9794;
   DATA[2365,14] := 1.0;
   DATA[2365,15] := 2.0;
   DATA[2365,16] := 1.0;
   DATA[2365,17] := 1.0;
   DATA[2365,18] := 1.0;
   DATA[2365,19] := 2.0;
   DATA[2365,20] := 148.808;
   DATA[2365,21] := 155.2166;
   DATA[2365,22] := 1.717874;
   DATA[2365,23] := 859.0105;
   DATA[2365,24] := 2.0;
   DATA[2365,25] := 2.0;
   DATA[2365,26] := 7.874135;
   DATA[2365,27] := 144.2194;
   DATA[2365,28] := 261.7278;
   DATA[2365,29] := 12.11228;
   DATA[2365,30] := 1.72443;
   DATA[2365,31] := 1.284745;
   DATA[2365,32] := 0.7353967;
   DATA[2365,33] := 0.3069532;
   DATA[2365,34] := 2.0;
   DATA[2365,35] := 250.1762;
   DATA[2365,36] := 1.762086;
   DATA[2365,37] := 188.9259;
   DATA[2365,38] := 0.000128152;
   DATA[2365,39] := 1.0;
   DATA[2365,40] := 1.0;
   DATA[2366,0] := 2.580469;
   DATA[2366,1] := 866.6616;
   DATA[2366,2] := 2.0;
   DATA[2366,3] := 2.0;
   DATA[2366,4] := 262.3366;
   DATA[2366,5] := 8.393232;
   DATA[2366,6] := 329.8898;
   DATA[2366,7] := 2.453337;
   DATA[2366,8] := 2.0;
   DATA[2366,9] := 2.0;
   DATA[2366,10] := 2.0;
   DATA[2366,11] := 19.68756;
   DATA[2366,12] := 2.209909;
   DATA[2366,13] := 817.9393;
   DATA[2366,14] := 1.0;
   DATA[2366,15] := 2.0;
   DATA[2366,16] := 1.0;
   DATA[2366,17] := 1.0;
   DATA[2366,18] := 1.0;
   DATA[2366,19] := 2.0;
   DATA[2366,20] := 148.808;
   DATA[2366,21] := 155.2166;
   DATA[2366,22] := 1.717874;
   DATA[2366,23] := 859.1643;
   DATA[2366,24] := 2.0;
   DATA[2366,25] := 2.0;
   DATA[2366,26] := 7.874135;
   DATA[2366,27] := 144.2194;
   DATA[2366,28] := 261.7278;
   DATA[2366,29] := 12.11228;
   DATA[2366,30] := 1.72443;
   DATA[2366,31] := 1.291533;
   DATA[2366,32] := 0.7353967;
   DATA[2366,33] := 0.3066329;
   DATA[2366,34] := 2.0;
   DATA[2366,35] := 250.1762;
   DATA[2366,36] := 1.762086;
   DATA[2366,37] := 188.9259;
   DATA[2366,38] := 0.000128152;
   DATA[2366,39] := 1.0;
   DATA[2366,40] := 1.0;
   DATA[2367,0] := 2.561253;
   DATA[2367,1] := 866.3869;
   DATA[2367,2] := 2.0;
   DATA[2367,3] := 2.0;
   DATA[2367,4] := 262.3366;
   DATA[2367,5] := 8.395475;
   DATA[2367,6] := 329.8898;
   DATA[2367,7] := 2.45449;
   DATA[2367,8] := 2.0;
   DATA[2367,9] := 2.0;
   DATA[2367,10] := 2.0;
   DATA[2367,11] := 19.65235;
   DATA[2367,12] := 2.209909;
   DATA[2367,13] := 817.9393;
   DATA[2367,14] := 1.0;
   DATA[2367,15] := 2.0;
   DATA[2367,16] := 1.0;
   DATA[2367,17] := 1.0;
   DATA[2367,18] := 1.0;
   DATA[2367,19] := 2.0;
   DATA[2367,20] := 148.808;
   DATA[2367,21] := 155.2166;
   DATA[2367,22] := 1.717874;
   DATA[2367,23] := 859.1643;
   DATA[2367,24] := 2.0;
   DATA[2367,25] := 2.0;
   DATA[2367,26] := 7.874135;
   DATA[2367,27] := 144.2194;
   DATA[2367,28] := 261.7278;
   DATA[2367,29] := 12.11228;
   DATA[2367,30] := 1.72443;
   DATA[2367,31] := 1.302293;
   DATA[2367,32] := 0.7353967;
   DATA[2367,33] := 0.3066329;
   DATA[2367,34] := 2.0;
   DATA[2367,35] := 250.1762;
   DATA[2367,36] := 1.681991;
   DATA[2367,37] := 188.9259;
   DATA[2367,38] := 0.000128152;
   DATA[2367,39] := 1.0;
   DATA[2367,40] := 1.0;
   DATA[2368,0] := 2.54684;
   DATA[2368,1] := 866.1514;
   DATA[2368,2] := 2.0;
   DATA[2368,3] := 2.0;
   DATA[2368,4] := 262.3366;
   DATA[2368,5] := 8.395475;
   DATA[2368,6] := 329.8898;
   DATA[2368,7] := 2.454875;
   DATA[2368,8] := 2.0;
   DATA[2368,9] := 2.0;
   DATA[2368,10] := 2.0;
   DATA[2368,11] := 19.64594;
   DATA[2368,12] := 2.209909;
   DATA[2368,13] := 817.4587;
   DATA[2368,14] := 1.0;
   DATA[2368,15] := 2.0;
   DATA[2368,16] := 1.0;
   DATA[2368,17] := 1.0;
   DATA[2368,18] := 1.0;
   DATA[2368,19] := 2.0;
   DATA[2368,20] := 148.808;
   DATA[2368,21] := 155.2166;
   DATA[2368,22] := 1.717874;
   DATA[2368,23] := 859.1259;
   DATA[2368,24] := 2.0;
   DATA[2368,25] := 2.0;
   DATA[2368,26] := 7.874135;
   DATA[2368,27] := 144.2194;
   DATA[2368,28] := 261.7278;
   DATA[2368,29] := 12.11228;
   DATA[2368,30] := 1.72443;
   DATA[2368,31] := 1.302293;
   DATA[2368,32] := 0.7353967;
   DATA[2368,33] := 0.3066329;
   DATA[2368,34] := 2.0;
   DATA[2368,35] := 250.1602;
   DATA[2368,36] := 1.681991;
   DATA[2368,37] := 188.9259;
   DATA[2368,38] := 0.000128152;
   DATA[2368,39] := 1.0;
   DATA[2368,40] := 1.0;
   DATA[2369,0] := 2.515453;
   DATA[2369,1] := 865.8766;
   DATA[2369,2] := 2.0;
   DATA[2369,3] := 2.0;
   DATA[2369,4] := 262.3366;
   DATA[2369,5] := 8.395475;
   DATA[2369,6] := 329.8898;
   DATA[2369,7] := 2.456156;
   DATA[2369,8] := 2.0;
   DATA[2369,9] := 2.0;
   DATA[2369,10] := 2.0;
   DATA[2369,11] := 19.69076;
   DATA[2369,12] := 2.209909;
   DATA[2369,13] := 817.0181;
   DATA[2369,14] := 1.0;
   DATA[2369,15] := 2.0;
   DATA[2369,16] := 1.0;
   DATA[2369,17] := 1.0;
   DATA[2369,18] := 1.0;
   DATA[2369,19] := 2.0;
   DATA[2369,20] := 148.808;
   DATA[2369,21] := 155.2166;
   DATA[2369,22] := 1.717874;
   DATA[2369,23] := 859.0105;
   DATA[2369,24] := 2.0;
   DATA[2369,25] := 2.0;
   DATA[2369,26] := 7.874135;
   DATA[2369,27] := 144.322;
   DATA[2369,28] := 261.7278;
   DATA[2369,29] := 12.11228;
   DATA[2369,30] := 1.72443;
   DATA[2369,31] := 1.29576;
   DATA[2369,32] := 0.7353967;
   DATA[2369,33] := 0.3066329;
   DATA[2369,34] := 2.0;
   DATA[2369,35] := 250.1442;
   DATA[2369,36] := 1.601897;
   DATA[2369,37] := 188.9259;
   DATA[2369,38] := 0.000128152;
   DATA[2369,39] := 1.0;
   DATA[2369,40] := 1.0;
   DATA[2370,0] := 2.502642;
   DATA[2370,1] := 865.5233;
   DATA[2370,2] := 2.0;
   DATA[2370,3] := 2.0;
   DATA[2370,4] := 262.3366;
   DATA[2370,5] := 8.395475;
   DATA[2370,6] := 329.8898;
   DATA[2370,7] := 2.456156;
   DATA[2370,8] := 2.0;
   DATA[2370,9] := 2.0;
   DATA[2370,10] := 2.0;
   DATA[2370,11] := 19.69076;
   DATA[2370,12] := 2.209909;
   DATA[2370,13] := 817.1783;
   DATA[2370,14] := 1.0;
   DATA[2370,15] := 2.0;
   DATA[2370,16] := 1.0;
   DATA[2370,17] := 1.0;
   DATA[2370,18] := 1.0;
   DATA[2370,19] := 2.0;
   DATA[2370,20] := 148.808;
   DATA[2370,21] := 155.2166;
   DATA[2370,22] := 1.717874;
   DATA[2370,23] := 858.7413;
   DATA[2370,24] := 2.0;
   DATA[2370,25] := 2.0;
   DATA[2370,26] := 7.874135;
   DATA[2370,27] := 144.322;
   DATA[2370,28] := 261.7278;
   DATA[2370,29] := 12.11228;
   DATA[2370,30] := 1.72443;
   DATA[2370,31] := 1.298194;
   DATA[2370,32] := 0.7353967;
   DATA[2370,33] := 0.3077859;
   DATA[2370,34] := 2.0;
   DATA[2370,35] := 250.1442;
   DATA[2370,36] := 1.601897;
   DATA[2370,37] := 188.9259;
   DATA[2370,38] := 0.000128152;
   DATA[2370,39] := 1.0;
   DATA[2370,40] := 1.0;
   DATA[2371,0] := 2.482785;
   DATA[2371,1] := 865.5233;
   DATA[2371,2] := 2.0;
   DATA[2371,3] := 2.0;
   DATA[2371,4] := 262.3366;
   DATA[2371,5] := 8.395475;
   DATA[2371,6] := 329.8898;
   DATA[2371,7] := 2.456412;
   DATA[2371,8] := 2.0;
   DATA[2371,9] := 2.0;
   DATA[2371,10] := 2.0;
   DATA[2371,11] := 19.69076;
   DATA[2371,12] := 2.209909;
   DATA[2371,13] := 817.0582;
   DATA[2371,14] := 1.0;
   DATA[2371,15] := 2.0;
   DATA[2371,16] := 1.0;
   DATA[2371,17] := 1.0;
   DATA[2371,18] := 1.0;
   DATA[2371,19] := 2.0;
   DATA[2371,20] := 148.808;
   DATA[2371,21] := 155.1653;
   DATA[2371,22] := 1.717874;
   DATA[2371,23] := 858.4337;
   DATA[2371,24] := 2.0;
   DATA[2371,25] := 2.0;
   DATA[2371,26] := 7.874135;
   DATA[2371,27] := 144.322;
   DATA[2371,28] := 261.7278;
   DATA[2371,29] := 12.11228;
   DATA[2371,30] := 1.72443;
   DATA[2371,31] := 1.285385;
   DATA[2371,32] := 0.7353967;
   DATA[2371,33] := 0.3081703;
   DATA[2371,34] := 2.0;
   DATA[2371,35] := 250.1442;
   DATA[2371,36] := 1.601897;
   DATA[2371,37] := 188.9259;
   DATA[2371,38] := 0.000128152;
   DATA[2371,39] := 1.0;
   DATA[2371,40] := 1.0;
   DATA[2372,0] := 2.469974;
   DATA[2372,1] := 865.6803;
   DATA[2372,2] := 2.0;
   DATA[2372,3] := 2.0;
   DATA[2372,4] := 262.3366;
   DATA[2372,5] := 8.395475;
   DATA[2372,6] := 329.8898;
   DATA[2372,7] := 2.456412;
   DATA[2372,8] := 2.0;
   DATA[2372,9] := 2.0;
   DATA[2372,10] := 2.0;
   DATA[2372,11] := 19.69076;
   DATA[2372,12] := 2.211318;
   DATA[2372,13] := 817.3385;
   DATA[2372,14] := 1.0;
   DATA[2372,15] := 2.0;
   DATA[2372,16] := 1.0;
   DATA[2372,17] := 1.0;
   DATA[2372,18] := 1.0;
   DATA[2372,19] := 2.0;
   DATA[2372,20] := 148.808;
   DATA[2372,21] := 155.1653;
   DATA[2372,22] := 1.717874;
   DATA[2372,23] := 858.5875;
   DATA[2372,24] := 2.0;
   DATA[2372,25] := 2.0;
   DATA[2372,26] := 7.874135;
   DATA[2372,27] := 144.322;
   DATA[2372,28] := 261.7278;
   DATA[2372,29] := 12.11228;
   DATA[2372,30] := 1.72443;
   DATA[2372,31] := 1.282183;
   DATA[2372,32] := 0.7353967;
   DATA[2372,33] := 0.3084265;
   DATA[2372,34] := 2.0;
   DATA[2372,35] := 250.0641;
   DATA[2372,36] := 1.601897;
   DATA[2372,37] := 188.9259;
   DATA[2372,38] := 0.000128152;
   DATA[2372,39] := 1.0;
   DATA[2372,40] := 1.0;
   DATA[2373,0] := 2.447555;
   DATA[2373,1] := 865.9551;
   DATA[2373,2] := 2.0;
   DATA[2373,3] := 2.0;
   DATA[2373,4] := 262.3366;
   DATA[2373,5] := 8.395475;
   DATA[2373,6] := 329.8898;
   DATA[2373,7] := 2.456412;
   DATA[2373,8] := 2.0;
   DATA[2373,9] := 2.0;
   DATA[2373,10] := 2.0;
   DATA[2373,11] := 19.66195;
   DATA[2373,12] := 2.212984;
   DATA[2373,13] := 817.0181;
   DATA[2373,14] := 1.0;
   DATA[2373,15] := 2.0;
   DATA[2373,16] := 1.0;
   DATA[2373,17] := 1.0;
   DATA[2373,18] := 1.0;
   DATA[2373,19] := 2.0;
   DATA[2373,20] := 148.808;
   DATA[2373,21] := 155.1653;
   DATA[2373,22] := 1.717874;
   DATA[2373,23] := 858.1261;
   DATA[2373,24] := 2.0;
   DATA[2373,25] := 2.0;
   DATA[2373,26] := 7.874135;
   DATA[2373,27] := 144.2194;
   DATA[2373,28] := 261.5355;
   DATA[2373,29] := 12.11228;
   DATA[2373,30] := 1.72443;
   DATA[2373,31] := 1.291149;
   DATA[2373,32] := 0.7353967;
   DATA[2373,33] := 0.3084265;
   DATA[2373,34] := 2.0;
   DATA[2373,35] := 249.9519;
   DATA[2373,36] := 1.681991;
   DATA[2373,37] := 188.9259;
   DATA[2373,38] := 0.000128152;
   DATA[2373,39] := 1.0;
   DATA[2373,40] := 1.0;
   DATA[2374,0] := 2.438267;
   DATA[2374,1] := 865.6803;
   DATA[2374,2] := 2.0;
   DATA[2374,3] := 2.0;
   DATA[2374,4] := 262.3366;
   DATA[2374,5] := 8.395475;
   DATA[2374,6] := 329.8129;
   DATA[2374,7] := 2.456412;
   DATA[2374,8] := 2.0;
   DATA[2374,9] := 2.0;
   DATA[2374,10] := 2.0;
   DATA[2374,11] := 19.66195;
   DATA[2374,12] := 2.212984;
   DATA[2374,13] := 817.1783;
   DATA[2374,14] := 1.0;
   DATA[2374,15] := 2.0;
   DATA[2374,16] := 1.0;
   DATA[2374,17] := 1.0;
   DATA[2374,18] := 1.0;
   DATA[2374,19] := 2.0;
   DATA[2374,20] := 148.808;
   DATA[2374,21] := 155.1653;
   DATA[2374,22] := 1.715439;
   DATA[2374,23] := 858.0107;
   DATA[2374,24] := 2.0;
   DATA[2374,25] := 2.0;
   DATA[2374,26] := 7.874135;
   DATA[2374,27] := 144.1169;
   DATA[2374,28] := 261.5355;
   DATA[2374,29] := 12.11228;
   DATA[2374,30] := 1.72443;
   DATA[2374,31] := 1.292046;
   DATA[2374,32] := 0.7353967;
   DATA[2374,33] := 0.3084265;
   DATA[2374,34] := 2.0;
   DATA[2374,35] := 249.9519;
   DATA[2374,36] := 1.681991;
   DATA[2374,37] := 188.9259;
   DATA[2374,38] := 0.000128152;
   DATA[2374,39] := 1.0;
   DATA[2374,40] := 1.0;
   DATA[2375,0] := 2.423854;
   DATA[2375,1] := 865.2093;
   DATA[2375,2] := 2.0;
   DATA[2375,3] := 2.0;
   DATA[2375,4] := 262.3366;
   DATA[2375,5] := 8.395475;
   DATA[2375,6] := 329.7103;
   DATA[2375,7] := 2.456412;
   DATA[2375,8] := 2.0;
   DATA[2375,9] := 2.0;
   DATA[2375,10] := 2.0;
   DATA[2375,11] := 19.68756;
   DATA[2375,12] := 2.212984;
   DATA[2375,13] := 817.1783;
   DATA[2375,14] := 1.0;
   DATA[2375,15] := 2.0;
   DATA[2375,16] := 1.0;
   DATA[2375,17] := 1.0;
   DATA[2375,18] := 1.0;
   DATA[2375,19] := 2.0;
   DATA[2375,20] := 148.808;
   DATA[2375,21] := 155.1653;
   DATA[2375,22] := 1.715439;
   DATA[2375,23] := 857.7416;
   DATA[2375,24] := 2.0;
   DATA[2375,25] := 2.0;
   DATA[2375,26] := 7.874135;
   DATA[2375,27] := 144.1169;
   DATA[2375,28] := 261.5355;
   DATA[2375,29] := 12.11228;
   DATA[2375,30] := 1.72443;
   DATA[2375,31] := 1.292046;
   DATA[2375,32] := 0.7353967;
   DATA[2375,33] := 0.3084265;
   DATA[2375,34] := 2.0;
   DATA[2375,35] := 249.9519;
   DATA[2375,36] := 1.681991;
   DATA[2375,37] := 188.9259;
   DATA[2375,38] := 0.000128152;
   DATA[2375,39] := 1.0;
   DATA[2375,40] := 1.0;
   DATA[2376,0] := 2.423854;
   DATA[2376,1] := 864.9738;
   DATA[2376,2] := 2.0;
   DATA[2376,3] := 2.0;
   DATA[2376,4] := 262.3366;
   DATA[2376,5] := 8.395475;
   DATA[2376,6] := 329.7103;
   DATA[2376,7] := 2.456412;
   DATA[2376,8] := 2.0;
   DATA[2376,9] := 2.0;
   DATA[2376,10] := 2.0;
   DATA[2376,11] := 19.69396;
   DATA[2376,12] := 2.211831;
   DATA[2376,13] := 817.1783;
   DATA[2376,14] := 1.0;
   DATA[2376,15] := 2.0;
   DATA[2376,16] := 1.0;
   DATA[2376,17] := 1.0;
   DATA[2376,18] := 1.0;
   DATA[2376,19] := 2.0;
   DATA[2376,20] := 148.808;
   DATA[2376,21] := 155.1653;
   DATA[2376,22] := 1.715439;
   DATA[2376,23] := 857.9723;
   DATA[2376,24] := 2.0;
   DATA[2376,25] := 2.0;
   DATA[2376,26] := 7.874135;
   DATA[2376,27] := 144.1169;
   DATA[2376,28] := 261.5355;
   DATA[2376,29] := 12.11228;
   DATA[2376,30] := 1.72443;
   DATA[2376,31] := 1.282439;
   DATA[2376,32] := 0.7353967;
   DATA[2376,33] := 0.3084265;
   DATA[2376,34] := 2.0;
   DATA[2376,35] := 249.9519;
   DATA[2376,36] := 1.681991;
   DATA[2376,37] := 188.9259;
   DATA[2376,38] := 0.000128152;
   DATA[2376,39] := 1.0;
   DATA[2376,40] := 1.0;
   DATA[2377,0] := 2.443071;
   DATA[2377,1] := 864.9738;
   DATA[2377,2] := 2.0;
   DATA[2377,3] := 2.0;
   DATA[2377,4] := 262.3366;
   DATA[2377,5] := 8.395475;
   DATA[2377,6] := 329.7103;
   DATA[2377,7] := 2.456412;
   DATA[2377,8] := 2.0;
   DATA[2377,9] := 2.0;
   DATA[2377,10] := 2.0;
   DATA[2377,11] := 19.69396;
   DATA[2377,12] := 2.211575;
   DATA[2377,13] := 817.1783;
   DATA[2377,14] := 1.0;
   DATA[2377,15] := 2.0;
   DATA[2377,16] := 1.0;
   DATA[2377,17] := 1.0;
   DATA[2377,18] := 1.0;
   DATA[2377,19] := 2.0;
   DATA[2377,20] := 148.808;
   DATA[2377,21] := 155.0628;
   DATA[2377,22] := 1.715439;
   DATA[2377,23] := 857.9723;
   DATA[2377,24] := 2.0;
   DATA[2377,25] := 2.0;
   DATA[2377,26] := 7.874135;
   DATA[2377,27] := 144.1169;
   DATA[2377,28] := 261.5355;
   DATA[2377,29] := 12.11228;
   DATA[2377,30] := 1.72443;
   DATA[2377,31] := 1.274241;
   DATA[2377,32] := 0.7353967;
   DATA[2377,33] := 0.3084265;
   DATA[2377,34] := 2.0;
   DATA[2377,35] := 249.9519;
   DATA[2377,36] := 1.681991;
   DATA[2377,37] := 188.9259;
   DATA[2377,38] := 0.000128152;
   DATA[2377,39] := 1.0;
   DATA[2377,40] := 1.0;
   DATA[2378,0] := 2.46549;
   DATA[2378,1] := 864.856;
   DATA[2378,2] := 2.0;
   DATA[2378,3] := 2.0;
   DATA[2378,4] := 262.3366;
   DATA[2378,5] := 8.395475;
   DATA[2378,6] := 329.7103;
   DATA[2378,7] := 2.455131;
   DATA[2378,8] := 2.0;
   DATA[2378,9] := 2.0;
   DATA[2378,10] := 2.0;
   DATA[2378,11] := 19.69396;
   DATA[2378,12] := 2.211575;
   DATA[2378,13] := 817.3385;
   DATA[2378,14] := 1.0;
   DATA[2378,15] := 2.0;
   DATA[2378,16] := 1.0;
   DATA[2378,17] := 1.0;
   DATA[2378,18] := 1.0;
   DATA[2378,19] := 2.0;
   DATA[2378,20] := 148.808;
   DATA[2378,21] := 155.0628;
   DATA[2378,22] := 1.71262;
   DATA[2378,23] := 857.8185;
   DATA[2378,24] := 2.0;
   DATA[2378,25] := 2.0;
   DATA[2378,26] := 7.874135;
   DATA[2378,27] := 144.1169;
   DATA[2378,28] := 261.5355;
   DATA[2378,29] := 12.11228;
   DATA[2378,30] := 1.72443;
   DATA[2378,31] := 1.271423;
   DATA[2378,32] := 0.7353967;
   DATA[2378,33] := 0.3084265;
   DATA[2378,34] := 2.0;
   DATA[2378,35] := 249.9519;
   DATA[2378,36] := 1.681991;
   DATA[2378,37] := 188.7977;
   DATA[2378,38] := 0.000128152;
   DATA[2378,39] := 1.0;
   DATA[2378,40] := 1.0;
   DATA[2379,0] := 2.525062;
   DATA[2379,1] := 864.856;
   DATA[2379,2] := 2.0;
   DATA[2379,3] := 2.0;
   DATA[2379,4] := 262.3366;
   DATA[2379,5] := 8.395475;
   DATA[2379,6] := 329.7103;
   DATA[2379,7] := 2.455131;
   DATA[2379,8] := 2.0;
   DATA[2379,9] := 2.0;
   DATA[2379,10] := 2.0;
   DATA[2379,11] := 19.62994;
   DATA[2379,12] := 2.210037;
   DATA[2379,13] := 817.5388;
   DATA[2379,14] := 1.0;
   DATA[2379,15] := 2.0;
   DATA[2379,16] := 1.0;
   DATA[2379,17] := 1.0;
   DATA[2379,18] := 1.0;
   DATA[2379,19] := 2.0;
   DATA[2379,20] := 148.808;
   DATA[2379,21] := 155.0628;
   DATA[2379,22] := 1.71262;
   DATA[2379,23] := 857.9338;
   DATA[2379,24] := 2.0;
   DATA[2379,25] := 2.0;
   DATA[2379,26] := 7.874135;
   DATA[2379,27] := 144.1938;
   DATA[2379,28] := 261.5355;
   DATA[2379,29] := 12.11228;
   DATA[2379,30] := 1.725711;
   DATA[2379,31] := 1.271423;
   DATA[2379,32] := 0.7353967;
   DATA[2379,33] := 0.3084265;
   DATA[2379,34] := 2.0;
   DATA[2379,35] := 249.9519;
   DATA[2379,36] := 1.681991;
   DATA[2379,37] := 188.7977;
   DATA[2379,38] := 0.000128152;
   DATA[2379,39] := 1.0;
   DATA[2379,40] := 1.0;
   DATA[2380,0] := 2.55773;
   DATA[2380,1] := 864.7383;
   DATA[2380,2] := 2.0;
   DATA[2380,3] := 2.0;
   DATA[2380,4] := 262.3366;
   DATA[2380,5] := 8.395475;
   DATA[2380,6] := 329.7103;
   DATA[2380,7] := 2.455131;
   DATA[2380,8] := 2.0;
   DATA[2380,9] := 2.0;
   DATA[2380,10] := 2.0;
   DATA[2380,11] := 19.57872;
   DATA[2380,12] := 2.209909;
   DATA[2380,13] := 817.6589;
   DATA[2380,14] := 1.0;
   DATA[2380,15] := 2.0;
   DATA[2380,16] := 1.0;
   DATA[2380,17] := 1.0;
   DATA[2380,18] := 1.0;
   DATA[2380,19] := 2.0;
   DATA[2380,20] := 148.808;
   DATA[2380,21] := 155.0628;
   DATA[2380,22] := 1.71262;
   DATA[2380,23] := 858.0492;
   DATA[2380,24] := 2.0;
   DATA[2380,25] := 2.0;
   DATA[2380,26] := 7.874135;
   DATA[2380,27] := 144.1938;
   DATA[2380,28] := 261.5355;
   DATA[2380,29] := 12.11228;
   DATA[2380,30] := 1.725711;
   DATA[2380,31] := 1.284873;
   DATA[2380,32] := 0.7353967;
   DATA[2380,33] := 0.3084265;
   DATA[2380,34] := 2.0;
   DATA[2380,35] := 249.9519;
   DATA[2380,36] := 1.681991;
   DATA[2380,37] := 188.7977;
   DATA[2380,38] := 0.000128152;
   DATA[2380,39] := 1.0;
   DATA[2380,40] := 1.0;
   DATA[2381,0] := 2.60481;
   DATA[2381,1] := 864.9345;
   DATA[2381,2] := 2.0;
   DATA[2381,3] := 2.0;
   DATA[2381,4] := 262.3366;
   DATA[2381,5] := 8.395475;
   DATA[2381,6] := 329.7103;
   DATA[2381,7] := 2.455131;
   DATA[2381,8] := 2.0;
   DATA[2381,9] := 2.0;
   DATA[2381,10] := 2.0;
   DATA[2381,11] := 19.57872;
   DATA[2381,12] := 2.209909;
   DATA[2381,13] := 817.5388;
   DATA[2381,14] := 1.0;
   DATA[2381,15] := 2.0;
   DATA[2381,16] := 1.0;
   DATA[2381,17] := 1.0;
   DATA[2381,18] := 1.0;
   DATA[2381,19] := 2.0;
   DATA[2381,20] := 148.808;
   DATA[2381,21] := 155.0628;
   DATA[2381,22] := 1.71262;
   DATA[2381,23] := 858.0492;
   DATA[2381,24] := 2.0;
   DATA[2381,25] := 2.0;
   DATA[2381,26] := 7.874135;
   DATA[2381,27] := 144.1938;
   DATA[2381,28] := 261.7278;
   DATA[2381,29] := 12.11228;
   DATA[2381,30] := 1.725711;
   DATA[2381,31] := 1.291277;
   DATA[2381,32] := 0.7353967;
   DATA[2381,33] := 0.3084265;
   DATA[2381,34] := 2.0;
   DATA[2381,35] := 250.0801;
   DATA[2381,36] := 1.681991;
   DATA[2381,37] := 188.7977;
   DATA[2381,38] := 0.000128152;
   DATA[2381,39] := 1.0;
   DATA[2381,40] := 1.0;
   DATA[2382,0] := 2.626909;
   DATA[2382,1] := 865.4056;
   DATA[2382,2] := 2.0;
   DATA[2382,3] := 2.0;
   DATA[2382,4] := 262.3366;
   DATA[2382,5] := 8.395475;
   DATA[2382,6] := 329.7103;
   DATA[2382,7] := 2.455131;
   DATA[2382,8] := 2.0;
   DATA[2382,9] := 2.0;
   DATA[2382,10] := 2.0;
   DATA[2382,11] := 19.57872;
   DATA[2382,12] := 2.209909;
   DATA[2382,13] := 817.7391;
   DATA[2382,14] := 1.0;
   DATA[2382,15] := 2.0;
   DATA[2382,16] := 1.0;
   DATA[2382,17] := 1.0;
   DATA[2382,18] := 1.0;
   DATA[2382,19] := 2.0;
   DATA[2382,20] := 148.808;
   DATA[2382,21] := 155.0628;
   DATA[2382,22] := 1.71262;
   DATA[2382,23] := 858.1261;
   DATA[2382,24] := 2.0;
   DATA[2382,25] := 2.0;
   DATA[2382,26] := 7.874135;
   DATA[2382,27] := 144.1938;
   DATA[2382,28] := 261.7278;
   DATA[2382,29] := 12.11228;
   DATA[2382,30] := 1.725711;
   DATA[2382,31] := 1.28705;
   DATA[2382,32] := 0.7353967;
   DATA[2382,33] := 0.3084265;
   DATA[2382,34] := 2.0;
   DATA[2382,35] := 250.0801;
   DATA[2382,36] := 1.681991;
   DATA[2382,37] := 188.7977;
   DATA[2382,38] := 0.000128152;
   DATA[2382,39] := 1.0;
   DATA[2382,40] := 1.0;
   DATA[2383,0] := 2.648048;
   DATA[2383,1] := 865.4841;
   DATA[2383,2] := 2.0;
   DATA[2383,3] := 2.0;
   DATA[2383,4] := 262.3366;
   DATA[2383,5] := 8.395475;
   DATA[2383,6] := 329.7103;
   DATA[2383,7] := 2.455131;
   DATA[2383,8] := 2.0;
   DATA[2383,9] := 2.0;
   DATA[2383,10] := 2.0;
   DATA[2383,11] := 19.66195;
   DATA[2383,12] := 2.208884;
